(* Global variable list: TwinCAT_Configuration *)
(* Generated automatically by TwinCAT - (read only) *)
VAR_CONFIG
	ST_Hydra8.a_signal_produktion AT %QX228.0 : BOOL;
	ST_Hydra8.a_signal_gutteil AT %QX228.1 : BOOL;
	ST_Hydra8.a_signal_schlechtteil AT %QX228.2 : BOOL;
	ST_Hydra8.a_signal_reserve AT %QX228.3 : BOOL;
	.ST00_170_Motorschutz.BitInToCheck AT %IX1204.0 : BOOL;	(*  ~ {LinkedWith:TIID^Gerät 2 (EtherCAT)^251_A1 (EK1100)^251_A10 (EL1809)^Channel 15^.ST00_170_Motorschutz.BitInToCheck} *)
	.ST00_170_Thermokont.BitInToCheck AT %IX1204.1 : BOOL;	(*  ~ {LinkedWith:TIID^Gerät 2 (EtherCAT)^251_A1 (EK1100)^251_A10 (EL1809)^Channel 16^.ST00_170_Thermokont.BitInToCheck} *)
	.ST00_245_V1.BitOutToSet AT %QX256.0 : BOOL;
	.ST00_245_V1.BitInToCheck AT %IX1412.0 : BOOL;
	.ST00_245_V2_START.BitOutToSet AT %QX256.1 : BOOL;
	.ST00_245_V2_START.BitInToCheck AT %IX1412.1 : BOOL;
	.ST00_245_V3_RESET.BitOutToSet AT %QX256.2 : BOOL;
	.ST00_245_V3_RESET.BitInToCheck AT %IX1412.2 : BOOL;
	.ST00_245_S1_STOP.BitInToCheck AT %IX1412.3 : BOOL;
	.ST00_245_S2_START.BitInToCheck AT %IX1412.4 : BOOL;
	.ST00_245_S3_RESET.BitInToCheck AT %IX1412.5 : BOOL;
	.ST00_72_K7.BitOutToSet AT %QX128.0 : BOOL;	(*  ~ {LinkedWith:TIID^Gerät 2 (EtherCAT)^251_A1 (EK1100)^252_A21 (EL2809)^Channel 4^.ST00_72_K7.BitOutToSet} *)
	.ST00_72_K7.BitInToCheck AT %IX1240.0 : BOOL;
	.ST00_73_K4.BitInToCheck AT %IX1388.0 : BOOL;	(*  ~ {LinkedWith:TIID^Gerät 2 (EtherCAT)^S1 A1 (EK1101)^DI1 (EL1004)^Channel 3^.ST00_73_K4.BitInToCheck AND.ST02_S1_40K01.BitInToCheck} *)
	.ST02_DT_95_A1.e_Ergebnis_iO AT %IX1240.2 : BOOL;	(*  ~ {LinkedWith:TIID^Gerät 2 (EtherCAT)^S1 A1 (EK1101)^DI4  (EL1809)^Channel 11^.ST02_DT_95_A1.e_Ergebnis_iO} *)
	.ST02_DT_95_A1.e_Ergebnis_niO AT %IX1240.3 : BOOL;	(*  ~ {LinkedWith:TIID^Gerät 2 (EtherCAT)^S1 A1 (EK1101)^DI4  (EL1809)^Channel 10^.ST02_DT_95_A1.e_Ergebnis_niO} *)
	.ST02_DT_95_A1.e_Betriebsbereit AT %IX1240.4 : BOOL;	(*  ~ {LinkedWith:TIID^Gerät 2 (EtherCAT)^S1 A1 (EK1101)^DI4  (EL1809)^Channel 9^.ST02_DT_95_A1.e_Betriebsbereit} *)
	.ST02_DT_95_A1.e_Best_Jobwechsel AT %IX1240.5 : BOOL;
	.ST02_DT_95_A1.a_Trigger AT %QX128.2 : BOOL;	(*  ~ {LinkedWith:TIID^Gerät 2 (EtherCAT)^S1 A1 (EK1101)^DO3 (EL2809)^Channel 6^.ST02_DT_95_A1.a_Trigger} *)
	.ST02_DT_95_A1.a_Job_Bit1 AT %QX128.3 : BOOL;	(*  ~ {LinkedWith:TIID^Gerät 2 (EtherCAT)^S1 A1 (EK1101)^DO3 (EL2809)^Channel 7^.ST02_DT_95_A1.a_Job_Bit1} *)
	.ST02_DT_95_A1.a_Job_Bit2 AT %QX128.4 : BOOL;	(*  ~ {LinkedWith:TIID^Gerät 2 (EtherCAT)^S1 A1 (EK1101)^DO3 (EL2809)^Channel 8^.ST02_DT_95_A1.a_Job_Bit2} *)
	.ST02_DT_95_A1.a_Job_Bit3 AT %QX196.0 : BOOL;
	.ST02_DT_95_A1.a_Job_Bit4 AT %QX196.1 : BOOL;
	.ST02_DT_95_A2.e_Betriebsbereit AT %IX1340.0 : BOOL;	(*  ~ {LinkedWith:TIID^Gerät 2 (EtherCAT)^S1 A1 (EK1101)^DI4  (EL1809)^Channel 9^.ST02_DT_95_A1.e_Betriebsbereit} *)
	.ST02_S1_66_B11.ValveSensor AT %IX1260.0 : BOOL;	(*  ~ {LinkedWith:TIID^Gerät 2 (EtherCAT)^DT_61A1(EP1816-0008)^DIG Inputs Channel 2^.ST02_S1_66_B11.ValveSensor} *)
	.ST02_S1_66_B21.ValveSensor AT %IX1260.1 : BOOL;	(*  ~ {LinkedWith:TIID^Gerät 2 (EtherCAT)^DT_61A1(EP1816-0008)^DIG Inputs Channel 2^.ST02_S1_66_B21.ValveSensor} *)
	.ST02_S1_66_B31.ValveSensor AT %IX1260.2 : BOOL;	(*  ~ {LinkedWith:TIID^Gerät 2 (EtherCAT)^DT_61A1(EP1816-0008)^DIG Inputs Channel 2^.ST02_S1_66_B31.ValveSensor} *)
	.ST02_S1_66_B41.ValveSensor AT %IX1260.3 : BOOL;	(*  ~ {LinkedWith:TIID^Gerät 2 (EtherCAT)^DT_61A1(EP1816-0008)^DIG Inputs Channel 2^.ST02_S1_66_B41.ValveSensor} *)
	.ST02_FDB_40_B61.BitInToCheck AT %IX1308.0 : BOOL;	(*  ~ {LinkedWith:TIID^Gerät 2 (EtherCAT)^S1 A1 (EK1101)^DI2 (EL1004)^Channel 1^.ST02_FDB_40_B61.BitInToCheck} *)
	.ST02_FDB_40_B71.BitInToCheck AT %IX1308.1 : BOOL;	(*  ~ {LinkedWith:TIID^Gerät 2 (EtherCAT)^S1 A1 (EK1101)^DI2 (EL1004)^Channel 2^.ST02_FDB_40_B71.BitInToCheck} *)
	.ST02_35_S31.BitInToCheck AT %IX1244.0 : BOOL;	(*  ~ {LinkedWith:TIID^Gerät 2 (EtherCAT)^S1 A1 (EK1101)^DI3 (EL1004)^Channel 4^.ST02_35_S31.BitInToCheck} *)
	.ST02_S1_6A01.BitInToCheck AT %IX1256.0 : BOOL;	(*  ~ {LinkedWith:TIID^Gerät 2 (EtherCAT)^S1 A1 (EK1101)^DI1 (EL1004)^Channel 1^.ST02_S1_6A01.BitInToCheck} *)
	.ST02_35Y01.CoilA AT %QX136.0 : BOOL;	(*  ~ {LinkedWith:TIID^Gerät 2 (EtherCAT)^S1 A1 (EK1101)^DO2 (EL2004)^Channel 1^.ST02_35Y01.CoilA} *)
	.ST02_35Y01.CoilB AT %QX136.1 : BOOL;
	.ST02_62_Y6.CoilA AT %QX148.0 : BOOL;	(*  ~ {LinkedWith:TIID^Gerät 2 (EtherCAT)^TDA_61A1 (CPX-FB38 64Byte)^Outputs^QB0^.ST02_62_Y6.CoilA} *)
	.ST02_62_Y6.CoilB AT %QX148.1 : BOOL;	(*  ~ {LinkedWith:TIID^Gerät 2 (EtherCAT)^TDA_61A1 (CPX-FB38 64Byte)^Outputs^QB0^.ST02_62_Y6.CoilB} *)
	.ST02_62_Y9.CoilA AT %QX144.0 : BOOL;	(*  ~ {LinkedWith:TIID^Gerät 2 (EtherCAT)^TDA_61A1 (CPX-FB38 64Byte)^Outputs^QB1^.ST02_62_Y9.CoilA} *)
	.ST02_62_Y9.CoilB AT %QX144.1 : BOOL;	(*  ~ {LinkedWith:TIID^Gerät 2 (EtherCAT)^TDA_61A1 (CPX-FB38 64Byte)^Outputs^QB1^.ST02_62_Y9.CoilB} *)
	.ST02_62_Y11.CoilA AT %QX144.2 : BOOL;	(*  ~ {LinkedWith:TIID^Gerät 2 (EtherCAT)^TDA_61A1 (CPX-FB38 64Byte)^Outputs^QB1^.ST02_62_Y11.CoilA} *)
	.ST02_62_Y11.CoilB AT %QX144.3 : BOOL;	(*  ~ {LinkedWith:TIID^Gerät 2 (EtherCAT)^TDA_61A1 (CPX-FB38 64Byte)^Outputs^QB1^.ST02_62_Y11.CoilB} *)
	.ST02_62_Y13.CoilA AT %QX144.4 : BOOL;	(*  ~ {LinkedWith:TIID^Gerät 2 (EtherCAT)^TDA_61A1 (CPX-FB38 64Byte)^Outputs^QB1^.ST02_62_Y13.CoilA} *)
	.ST02_62_Y13.CoilB AT %QX144.5 : BOOL;	(*  ~ {LinkedWith:TIID^Gerät 2 (EtherCAT)^TDA_61A1 (CPX-FB38 64Byte)^Outputs^QB1^.ST02_62_Y13.CoilB} *)
	.ST02_62_Y15.CoilA AT %QX144.6 : BOOL;	(*  ~ {LinkedWith:TIID^Gerät 2 (EtherCAT)^TDA_61A1 (CPX-FB38 64Byte)^Outputs^QB1^.ST02_62_Y15.CoilA} *)
	.ST02_62_Y15.CoilB AT %QX144.7 : BOOL;	(*  ~ {LinkedWith:TIID^Gerät 2 (EtherCAT)^TDA_61A1 (CPX-FB38 64Byte)^Outputs^QB1^.ST02_62_Y15.CoilB} *)
	.ST02_62_Y17.CoilA AT %QX145.0 : BOOL;	(*  ~ {LinkedWith:TIID^Gerät 2 (EtherCAT)^TDA_61A1 (CPX-FB38 64Byte)^Outputs^QB2^.ST02_62_Y17.CoilA} *)
	.ST02_62_Y17.CoilB AT %QX145.1 : BOOL;
	.ST02_62_Y18.CoilA AT %QX145.2 : BOOL;	(*  ~ {LinkedWith:TIID^Gerät 2 (EtherCAT)^TDA_61A1 (CPX-FB38 64Byte)^Outputs^QB2^.ST02_62_Y18.CoilA} *)
	.ST02_62_Y18.CoilB AT %QX145.3 : BOOL;
	.ST03_51_M1.e_Position AT %IB1312 : UDINT;	(*  ~ {LinkedWith:TIID^Gerät 2 (EtherCAT)^251_A1 (EK1100)^252_PM1(EL7211-0010)^FB Position^.ST03_51_M1.e_Position} *)
	.ST03_51_M1.e_Statusword AT %IB1316 : UINT;	(*  ~ {LinkedWith:TIID^Gerät 2 (EtherCAT)^251_A1 (EK1100)^252_PM1(EL7211-0010)^DRV Statusword^.ST03_51_M1.e_Statusword} *)
	.ST03_51_M1.e_Velocity AT %IB1318 : DINT;	(*  ~ {LinkedWith:TIID^Gerät 2 (EtherCAT)^251_A1 (EK1100)^252_PM1(EL7211-0010)^DRV Velocity actual value^.ST03_51_M1.e_Velocity} *)
	.ST03_51_M1.e_Torque AT %IB1328 : INT;
	.ST03_51_M1.e_Following_Error AT %IB1322 : DINT;	(*  ~ {LinkedWith:TIID^Gerät 2 (EtherCAT)^251_A1 (EK1100)^252_PM1(EL7211-0010)^DRV Following error actual value^.ST03_51_M1.e_Following_Error} *)
	.ST03_51_M1.e_Toggle AT %IX1326.0 : BOOL;	(*  ~ {LinkedWith:TIID^Gerät 2 (EtherCAT)^251_A1 (EK1100)^252_PM1(EL7211-0010)^WcState^InputToggle} *)
	.ST03_51_M1.e_State AT %IB1377 : UINT;
	.ST03_51_M1.a_Controlword AT %QB176 : UINT;	(*  ~ {LinkedWith:TIID^Gerät 2 (EtherCAT)^251_A1 (EK1100)^252_PM1(EL7211-0010)^DRV Controlword^.ST03_51_M1.a_Controlword} *)
	.ST03_51_M1.a_Target_Velocity AT %QB178 : DINT;	(*  ~ {LinkedWith:TIID^Gerät 2 (EtherCAT)^251_A1 (EK1100)^252_PM1(EL7211-0010)^DRV Target velocity^.ST03_51_M1.a_Target_Velocity} *)
	.ST03_51_M1.a_Target_Position AT %QB182 : UDINT;	(*  ~ {LinkedWith:TIID^Gerät 2 (EtherCAT)^251_A1 (EK1100)^252_PM1(EL7211-0010)^DRV Target position^.ST03_51_M1.a_Target_Position} *)
	.ST03_601V1_A1.BitOutToSet AT %QX228.4 : BOOL;
	.ST03_601V1_A1.BitInToCheck AT %IX1379.0 : BOOL;
	.Robot01.CollisionSensor AT %IX1379.1 : BOOL;
	.ST03_BG3_X53_0.BitInToCheck AT %IX1340.1 : BOOL;
	.ST03_65_Q1.BitOutToSet AT %QX252.0 : BOOL;
	.ST03_65_Q1.BitInToCheck AT %IX1408.0 : BOOL;
	.ST03_65_F1.BitInToCheck AT %IX1408.1 : BOOL;
	.ST03_8_100_A1.e_Betriebsbereit AT %IX1412.6 : BOOL;
	.ST03_8_103_A1.e_Betriebsbereit AT %IX1480.0 : BOOL;
	.ST03_418_B60_0.ValveSensor AT %IX1296.0 : BOOL;
	.ST03_418_B60_1.ValveSensor AT %IX1296.1 : BOOL;
	.ST03_418_B60_2.ValveSensor AT %IX1296.2 : BOOL;
	.ST03_418_B60_3.ValveSensor AT %IX1296.3 : BOOL;
	.ST03_418_B60_4.ValveSensor AT %IX1296.4 : BOOL;
	.ST03_418_B60_5.ValveSensor AT %IX1296.5 : BOOL;
	.ST03_418_B60_6.BitInToCheck AT %IX1296.6 : BOOL;
	.ST03_418_B60_7.BitInToCheck AT %IX1296.7 : BOOL;
	.ST03_419_B61_0.BitInToCheck AT %IX1297.0 : BOOL;
	.ST03_419_B61_1.BitInToCheck AT %IX1297.1 : BOOL;
	.ST03_419_B61_2.BitInToCheck AT %IX1297.2 : BOOL;
	.ST03_419_B61_3.BitInToCheck AT %IX1297.3 : BOOL;
	.ST03_419_Y61_5.CoilA AT %QX172.0 : BOOL;
	.ST03_419_Y61_5.CoilB AT %QX172.1 : BOOL;
	.ST03_419_Y61_6.CoilA AT %QX172.2 : BOOL;
	.ST03_419_Y61_6.CoilB AT %QX172.3 : BOOL;
	.ST03_419_Y61_7.CoilA AT %QX172.4 : BOOL;
	.ST03_419_Y61_7.CoilB AT %QX172.5 : BOOL;
	.ST03_425_B67_0.ValveSensor AT %IX1330.0 : BOOL;
	.ST03_425_B67_1.ValveSensor AT %IX1330.1 : BOOL;
	.ST03_425_B67_2.ValveSensor AT %IX1330.2 : BOOL;
	.ST03_425_B67_3.ValveSensor AT %IX1330.3 : BOOL;
	.ST03_425_B67_4.BitInToCheck AT %IX1330.4 : BOOL;
	.ST03_425_B67_5.BitInToCheck AT %IX1330.5 : BOOL;
	.ST03_425_B67_6.BitInToCheck AT %IX1330.6 : BOOL;
	.ST03_425_B67_7.BitInToCheck AT %IX1330.7 : BOOL;
	.ST03_426_B68_4.BitInToCheck AT %IX1331.0 : BOOL;
	.ST03_426_Y68_5.CoilA AT %QX188.0 : BOOL;
	.ST03_426_Y68_5.CoilB AT %QX188.1 : BOOL;
	.ST03_426_Y68_6.CoilA AT %QX188.2 : BOOL;
	.ST03_426_Y68_6.CoilB AT %QX188.3 : BOOL;
	.ST03_421_B63_0.ValveSensor AT %IX1297.4 : BOOL;
	.ST03_421_B63_1.ValveSensor AT %IX1297.5 : BOOL;
	.ST03_421_B63_2.ValveSensor AT %IX1297.6 : BOOL;
	.ST03_421_B63_3.ValveSensor AT %IX1297.7 : BOOL;
	.ST03_421_B63_4.BitInToCheck AT %IX1298.0 : BOOL;
	.ST03_421_B63_5.BitInToCheck AT %IX1298.1 : BOOL;
	.ST03_421_B63_6.BitInToCheck AT %IX1298.2 : BOOL;
	.ST03_421_B63_7.BitInToCheck AT %IX1298.3 : BOOL;
	.ST03_422_B64_0.BitInToCheck AT %IX1298.4 : BOOL;
	.ST03_423_B66_0.BitInToCheck AT %IX1340.2 : BOOL;
	.ST03_8_B76_1.BitInToCheck AT %IX1340.3 : BOOL;
	.ST03_8_B76_2.BitInToCheck AT %IX1340.4 : BOOL;
	.ST03_422_B64_1.ValveSensor AT %IX1298.5 : BOOL;
	.ST03_422_B64_2.ValveSensor AT %IX1298.6 : BOOL;
	.ST03_422_B64_3.BitInToCheck AT %IX1298.7 : BOOL;
	.ST03_422_B64_4.BitInToCheck AT %IX1299.0 : BOOL;
	.ST03_422_Y64_5.CoilA AT %QX172.6 : BOOL;
	.ST03_422_Y64_5.CoilB AT %QX172.7 : BOOL;
	.ST03_422_Y64_6.CoilA AT %QX173.0 : BOOL;
	.ST03_422_Y64_6.CoilB AT %QX173.1 : BOOL;
	.ST03_422_Y64_7.CoilA AT %QX173.2 : BOOL;
	.ST03_422_Y64_7.CoilB AT %QX173.3 : BOOL;
	.ST03_423_B65_0.ValveSensor AT %IX1340.5 : BOOL;
	.ST03_423_B65_1.ValveSensor AT %IX1340.6 : BOOL;
	.ST03_423_B65_2.BitInToCheck AT %IX1340.7 : BOOL;
	.ST03_423_B65_3.ValveSensor AT %IX1341.0 : BOOL;
	.ST03_423_B65_4.ValveSensor AT %IX1341.1 : BOOL;
	.ST03_423_B65_5.BitInToCheck AT %IX1341.2 : BOOL;
	.ST03_423_Y65_6.CoilA AT %QX196.2 : BOOL;
	.ST03_423_Y65_6.CoilB AT %QX196.3 : BOOL;
	.ST03_423_Y65_7.CoilA AT %QX196.4 : BOOL;
	.ST03_423_Y65_7.CoilB AT %QX196.5 : BOOL;
	.ST03_33F4.BitInToCheck AT %IX1299.1 : BOOL;
	.ST03_70U3_1.BitInToCheck AT %IX1299.2 : BOOL;
	.ST03_70U3_2.BitInToCheck AT %IX1299.3 : BOOL;
	.ST03_70U3_3.BitInToCheck AT %IX1299.4 : BOOL;
	.ST03_71U3_1.BitInToCheck AT %IX1299.5 : BOOL;
	.ST03_71U3_2.BitInToCheck AT %IX1299.6 : BOOL;
	.ST03_71U3_3.BitInToCheck AT %IX1299.7 : BOOL;
	.ST03_8_80_A1.e_Ergebnis_iO AT %IX1300.0 : BOOL;
	.ST03_8_80_A1.e_Ergebnis_niO AT %IX1300.1 : BOOL;
	.ST03_8_80_A1.e_Betriebsbereit AT %IX1300.2 : BOOL;
	.ST03_8_80_A1.e_Best_Jobwechsel AT %IX1300.3 : BOOL;
	.ST03_8_80_A1.a_Trigger AT %QX173.4 : BOOL;
	.ST03_8_80_A1.a_Job_Bit1 AT %QX173.5 : BOOL;
	.ST03_8_80_A1.a_Job_Bit2 AT %QX173.6 : BOOL;
	.ST03_8_80_A1.a_Job_Bit3 AT %QX196.6 : BOOL;
	.ST03_8_80_A1.a_Job_Bit4 AT %QX196.7 : BOOL;
	.ST03_8_85_A1.e_Ergebnis_iO AT %IX1300.4 : BOOL;
	.ST03_8_85_A1.e_Ergebnis_niO AT %IX1300.5 : BOOL;
	.ST03_8_85_A1.e_Betriebsbereit AT %IX1300.6 : BOOL;
	.ST03_8_85_A1.e_Best_Jobwechsel AT %IX1300.7 : BOOL;
	.ST03_8_85_A1.a_Trigger AT %QX173.7 : BOOL;
	.ST03_8_85_A1.a_Job_Bit1 AT %QX174.0 : BOOL;
	.ST03_8_85_A1.a_Job_Bit2 AT %QX174.1 : BOOL;
	.ST03_8_85_A1.a_Job_Bit3 AT %QX197.0 : BOOL;
	.ST03_8_85_A1.a_Job_Bit4 AT %QX197.1 : BOOL;
	.ST03_8_90_A1.e_Betriebsbereit AT %IX1341.3 : BOOL;
	.ST03_8_95_A1.e_Betriebsbereit AT %IX1341.4 : BOOL;
	.ST03_PLAN_70V1_1.BitOutToSet AT %QX174.2 : BOOL;
	.ST03_PLAN_70V1_1.BitInToCheck AT %IX1301.0 : BOOL;
	.ST03_PLAN_71V1_2.BitOutToSet AT %QX174.3 : BOOL;
	.ST03_PLAN_71V1_2.BitInToCheck AT %IX1301.1 : BOOL;
	.ST03_Y01.CoilA AT %QX197.2 : BOOL;
	.ST03_Y01.CoilB AT %QX197.3 : BOOL;
	.ST03_S18.BitInToCheck AT %IX1341.5 : BOOL;
	.ST03_435_B67_0.ValveSensor AT %IX1336.0 : BOOL;
	.ST03_435_B67_1.ValveSensor AT %IX1336.1 : BOOL;
	.ST03_435_B67_2.ValveSensor AT %IX1336.2 : BOOL;
	.ST03_435_B67_3.ValveSensor AT %IX1336.3 : BOOL;
	.ST03_435_B67_4.BitInToCheck AT %IX1336.4 : BOOL;
	.ST03_435_B67_7.BitInToCheck AT %IX1336.5 : BOOL;
	.ST03_436_B68_1.BitInToCheck AT %IX1336.6 : BOOL;
	.ST03_436_B68_2.BitInToCheck AT %IX1336.7 : BOOL;
	.ST03_437_B68_3.BitInToCheck AT %IX1337.0 : BOOL;
	.ST03_437_B68_4.BitInToCheck AT %IX1337.1 : BOOL;
	.ST03_437_Y68_5.CoilA AT %QX192.0 : BOOL;
	.ST03_437_Y68_5.CoilB AT %QX192.1 : BOOL;
	.ST03_437_Y68_6.CoilA AT %QX192.2 : BOOL;
	.ST03_437_Y68_6.CoilB AT %QX192.3 : BOOL;
	.ST03_444_B69_0.ValveSensor AT %IX1341.6 : BOOL;
	.ST03_444_B69_1.ValveSensor AT %IX1341.7 : BOOL;
	.ST03_444_B69_2.ValveSensor AT %IX1342.0 : BOOL;
	.ST03_444_B69_3.ValveSensor AT %IX1342.1 : BOOL;
	.ST03_444_B69_4.BitInToCheck AT %IX1342.2 : BOOL;
	.ST03_444_B69_7.BitInToCheck AT %IX1342.3 : BOOL;
	.ST03_445_B70_1.BitInToCheck AT %IX1342.4 : BOOL;
	.ST03_445_B70_2.BitInToCheck AT %IX1342.5 : BOOL;
	.ST03_446_B70_3.BitInToCheck AT %IX1342.6 : BOOL;
	.ST03_446_B70_4.BitInToCheck AT %IX1342.7 : BOOL;
	.ST03_446_Y70_5.CoilA AT %QX197.4 : BOOL;
	.ST03_446_Y70_5.CoilB AT %QX197.5 : BOOL;
	.ST03_446_Y70_6.CoilA AT %QX197.6 : BOOL;
	.ST03_446_Y70_6.CoilB AT %QX197.7 : BOOL;
	.ST03_451_B69_0.ValveSensor AT %IX1344.0 : BOOL;
	.ST03_451_B69_1.ValveSensor AT %IX1344.1 : BOOL;
	.ST03_451_B69_2.ValveSensor AT %IX1344.2 : BOOL;
	.ST03_451_B69_3.ValveSensor AT %IX1344.3 : BOOL;
	.ST03_451_B69_4.BitInToCheck AT %IX1344.4 : BOOL;
	.ST03_451_B69_7.BitInToCheck AT %IX1344.5 : BOOL;
	.ST03_452_B70_1.BitInToCheck AT %IX1344.6 : BOOL;
	.ST03_452_B70_2.BitInToCheck AT %IX1344.7 : BOOL;
	.ST03_453_B70_3.BitInToCheck AT %IX1345.0 : BOOL;
	.ST03_453_B70_4.BitInToCheck AT %IX1345.1 : BOOL;
	.ST03_453_Y70_5.CoilA AT %QX204.0 : BOOL;
	.ST03_453_Y70_5.CoilB AT %QX204.1 : BOOL;
	.ST03_453_Y70_6.CoilA AT %QX204.2 : BOOL;
	.ST03_453_Y70_6.CoilB AT %QX204.3 : BOOL;
	.ST03_461_B69_0.ValveSensor AT %IX1364.1 : BOOL;
	.ST03_461_B69_1.ValveSensor AT %IX1364.2 : BOOL;
	.ST03_461_B69_2.ValveSensor AT %IX1364.3 : BOOL;
	.ST03_461_B69_3.ValveSensor AT %IX1364.4 : BOOL;
	.ST03_461_B69_4.BitInToCheck AT %IX1364.5 : BOOL;
	.ST03_461_B69_5.ValveSensor AT %IX1364.6 : BOOL;
	.ST03_461_B69_6.ValveSensor AT %IX1364.7 : BOOL;
	.ST03_461_B69_7.BitInToCheck AT %IX1365.0 : BOOL;
	.ST03_462_B70_0.BitInToCheck AT %IX1365.1 : BOOL;
	.ST03_462_B70_1.BitInToCheck AT %IX1365.2 : BOOL;
	.ST03_462_B70_2.BitInToCheck AT %IX1365.3 : BOOL;
	.ST03_463_B70_3.ValveSensor AT %IX1365.4 : BOOL;
	.ST03_463_B70_4.ValveSensor AT %IX1365.5 : BOOL;
	.ST03_463_B70_5.ValveSensor AT %IX1365.6 : BOOL;
	.ST03_463_B70_6.ValveSensor AT %IX1365.7 : BOOL;
	.ST03_463_B70_7.BitInToCheck AT %IX1366.0 : BOOL;
	.ST03_464_Y71_0.CoilA AT %QX218.0 : BOOL;
	.ST03_464_Y71_0.CoilB AT %QX218.1 : BOOL;
	.ST03_464_Y71_1.CoilA AT %QX218.2 : BOOL;
	.ST03_464_Y71_1.CoilB AT %QX218.3 : BOOL;
	.ST03_464_Y71_2.CoilA AT %QX218.4 : BOOL;
	.ST03_464_Y71_2.CoilB AT %QX218.5 : BOOL;
	.ST03_464_Y71_3.CoilA AT %QX218.6 : BOOL;
	.ST03_464_Y71_3.CoilB AT %QX218.7 : BOOL;
	.ST03_464_Y71_4.CoilA AT %QX219.0 : BOOL;
	.ST03_464_Y71_4.CoilB AT %QX219.1 : BOOL;
	.ST03_464_Y71_5.CoilA AT %QX219.2 : BOOL;
	.ST03_464_Y71_5.CoilB AT %QX219.3 : BOOL;
	.ST03_464_B71_6.BitInToCheck AT %IX1366.1 : BOOL;
	.ST03_464_B71_7.BitInToCheck AT %IX1366.2 : BOOL;
	.ST03_8_105_A1.anInputRequest AT %QB288 : ARRAY [0..4] OF DWORD;
	.ST03_8_105_A1.bError_Status_00 AT %IX1464.0 : BOOL;
	.ST03_8_105_A1.bChange_Program_Ack AT %IX1464.1 : BOOL;
	.ST03_8_105_A1.bChange_Program_Failed AT %IX1464.2 : BOOL;
	.ST03_8_105_A1.bTotal_Status_OK_01 AT %IX1464.3 : BOOL;
	.ST03_8_105_A1.bTotal_Status_NG AT %IX1464.4 : BOOL;
	.ST03_8_105_A1.bRun AT %IX1464.5 : BOOL;
	.ST03_8_105_A1.bBusy AT %IX1464.6 : BOOL;
	.ST03_8_105_A1.bTrigger_Ready AT %IX1464.7 : BOOL;
	.ST03_8_105_A1.bTrigger_Ack AT %IX1465.0 : BOOL;
	.ST03_8_105_A1.abProgram_Num AT %IB1466 : ARRAY [0..6] OF BOOL;
	.ST03_8_105_A1.nState AT %IB1473 : UINT;
	.ST03_4x2_B69_0.BitInToCheck AT %IX1366.3 : BOOL;
	.ST03_4x2_B69_1.ValveSensor AT %IX1366.4 : BOOL;
	.ST03_4x2_B69_2.ValveSensor AT %IX1366.5 : BOOL;
	.ST03_4x2_B69_3.ValveSensor AT %IX1366.6 : BOOL;
	.ST03_4x2_B69_4.ValveSensor AT %IX1366.7 : BOOL;
	.ST03_4x2_B69_5.BitInToCheck AT %IX1392.0 : BOOL;
	.ST03_4x2_B69_6.ValveSensor AT %IX1367.1 : BOOL;
	.ST03_4x2_B69_7.ValveSensor AT %IX1392.1 : BOOL;
	.ST03_4x3_B70_0.BitInToCheck AT %IX1367.3 : BOOL;
	.ST03_4x3_B70_1.BitInToCheck AT %IX1392.2 : BOOL;
	.ST03_4x3_Y70_5.CoilA AT %QX236.0 : BOOL;
	.ST03_4x3_Y70_5.CoilB AT %QX236.1 : BOOL;
	.ST03_4x3_Y70_6.CoilA AT %QX236.2 : BOOL;
	.ST03_4x3_Y70_6.CoilB AT %QX236.3 : BOOL;
	.ST03_4x3_Y70_7.CoilA AT %QX236.4 : BOOL;
	.ST03_4x3_Y70_7.CoilB AT %QX236.5 : BOOL;
	.ST03_491_B69_0.BitInToCheck AT %IX1372.0 : BOOL;
	.ST03_491_B69_1.ValveSensor AT %IX1372.1 : BOOL;
	.ST03_491_B69_2.ValveSensor AT %IX1372.2 : BOOL;
	.ST03_491_B69_3.ValveSensor AT %IX1372.3 : BOOL;
	.ST03_491_B69_4.ValveSensor AT %IX1372.4 : BOOL;
	.ST03_491_B69_5.BitInToCheck AT %IX1372.5 : BOOL;
	.ST03_491_B69_7.BitInToCheck AT %IX1372.6 : BOOL;
	.ST03_492_Y70_0.CoilA AT %QX224.0 : BOOL;
	.ST03_492_Y70_0.CoilB AT %QX224.1 : BOOL;
	.ST03_492_Y70_1.CoilA AT %QX224.2 : BOOL;
	.ST03_492_Y70_1.CoilB AT %QX224.3 : BOOL;
	.ST03_501_B69_0.BitInToCheck AT %IX1379.4 : BOOL;
	.ST03_501_B69_1.ValveSensor AT %IX1379.5 : BOOL;
	.ST03_501_B69_2.ValveSensor AT %IX1379.6 : BOOL;
	.ST03_501_B69_3.ValveSensor AT %IX1379.7 : BOOL;
	.ST03_501_B69_4.ValveSensor AT %IX1380.0 : BOOL;
	.ST03_501_B69_5.BitInToCheck AT %IX1380.1 : BOOL;
	.ST03_501_B69_6.BitInToCheck AT %IX1380.2 : BOOL;
	.ST03_501_B69_7.BitInToCheck AT %IX1380.3 : BOOL;
	.ST03_502_B70_0.BitInToCheck AT %IX1380.4 : BOOL;
	.ST03_502_Y70_1.CoilA AT %QX228.7 : BOOL;
	.ST03_502_Y70_1.CoilB AT %QX229.0 : BOOL;
	.ST03_502_Y70_2.CoilA AT %QX229.1 : BOOL;
	.ST03_502_Y70_2.CoilB AT %QX229.2 : BOOL;
	.ST03_521_B69_0.BitInToCheck AT %IX1392.3 : BOOL;
	.ST03_521_B69_1.ValveSensor AT %IX1392.4 : BOOL;
	.ST03_521_B69_2.ValveSensor AT %IX1392.5 : BOOL;
	.ST03_521_B69_3.ValveSensor AT %IX1392.6 : BOOL;
	.ST03_521_B69_4.ValveSensor AT %IX1392.7 : BOOL;
	.ST03_521_B69_6.BitInToCheck AT %IX1393.0 : BOOL;
	.ST03_521_B69_7.BitInToCheck AT %IX1393.1 : BOOL;
	.ST03_522_B70_0.BitInToCheck AT %IX1393.2 : BOOL;
	.ST03_522_Y70_1.CoilA AT %QX236.6 : BOOL;
	.ST03_522_Y70_1.CoilB AT %QX236.7 : BOOL;
	.ST03_522_Y70_2.CoilA AT %QX237.0 : BOOL;
	.ST03_522_Y70_2.CoilB AT %QX237.1 : BOOL;
	.ST03_512_XG1.BitInToCheck AT %IX1380.5 : BOOL;	(*  ~ {LinkedWith:TIID^Gerät 2 (EtherCAT)^930_A2 (EP2338-0001)^Channel 1^.ST03_512_XG1.BitInToCheck} *)
	.ST03_512_B69_1.ValveSensor AT %IX1380.6 : BOOL;	(*  ~ {LinkedWith:TIID^Gerät 2 (EtherCAT)^930_A2 (EP2338-0001)^Channel 2^.ST03_512_B69_1.ValveSensor} *)
	.ST03_512_B69_2.ValveSensor AT %IX1380.7 : BOOL;	(*  ~ {LinkedWith:TIID^Gerät 2 (EtherCAT)^930_A2 (EP2338-0001)^Channel 3^.ST03_512_B69_2.ValveSensor} *)
	.ST03_512_B69_3.ValveSensor AT %IX1381.0 : BOOL;	(*  ~ {LinkedWith:TIID^Gerät 2 (EtherCAT)^930_A2 (EP2338-0001)^Channel 4^.ST03_512_B69_3.ValveSensor} *)
	.ST03_512_B69_4.ValveSensor AT %IX1381.1 : BOOL;	(*  ~ {LinkedWith:TIID^Gerät 2 (EtherCAT)^930_A2 (EP2338-0001)^Channel 5^.ST03_512_B69_4.ValveSensor} *)
	.ST03_512_B69_5.ValveSensor AT %IX1388.1 : BOOL;	(*  ~ {LinkedWith:TIID^Gerät 2 (EtherCAT)^930_A2 (EP2338-0001)^Channel 6^.ST03_512_B69_5.ValveSensor} *)
	.ST03_512_B69_6.ValveSensor AT %IX1388.2 : BOOL;	(*  ~ {LinkedWith:TIID^Gerät 2 (EtherCAT)^930_A2 (EP2338-0001)^Channel 7^.ST03_512_B69_6.ValveSensor} *)
	.ST03_513_B70_0.ValveSensor AT %IX1381.3 : BOOL;	(*  ~ {LinkedWith:TIID^Gerät 2 (EtherCAT)^931_A3 (EP2338-0001)^Channel 1^.ST03_513_B70_0.ValveSensor} *)
	.ST03_513_B70_1.ValveSensor AT %IX1381.4 : BOOL;	(*  ~ {LinkedWith:TIID^Gerät 2 (EtherCAT)^931_A3 (EP2338-0001)^Channel 2^.ST03_513_B70_1.ValveSensor} *)
	.ST03_513_B70_2.ValveSensor AT %IX1381.5 : BOOL;	(*  ~ {LinkedWith:TIID^Gerät 2 (EtherCAT)^931_A3 (EP2338-0001)^Channel 3^.ST03_513_B70_2.ValveSensor} *)
	.ST03_513_B70_3.ValveSensor AT %IX1381.6 : BOOL;	(*  ~ {LinkedWith:TIID^Gerät 2 (EtherCAT)^931_A3 (EP2338-0001)^Channel 4^.ST03_513_B70_3.ValveSensor} *)
	.ST03_513_B70_4.BitInToCheck AT %IX1381.7 : BOOL;	(*  ~ {LinkedWith:TIID^Gerät 2 (EtherCAT)^931_A3 (EP2338-0001)^Channel 5^.ST03_513_B70_4.BitInToCheck} *)
	.ST03_513_B70_5.ValveSensor AT %IX1382.0 : BOOL;	(*  ~ {LinkedWith:TIID^Gerät 2 (EtherCAT)^931_A3 (EP2338-0001)^Channel 6^.ST03_513_B70_5.ValveSensor} *)
	.ST03_513_B70_6.ValveSensor AT %IX1382.1 : BOOL;	(*  ~ {LinkedWith:TIID^Gerät 2 (EtherCAT)^931_A3 (EP2338-0001)^Channel 7^.ST03_513_B70_6.ValveSensor} *)
	.ST03_513_B70_7.BitInToCheck AT %IX1382.2 : BOOL;	(*  ~ {LinkedWith:TIID^Gerät 2 (EtherCAT)^931_A3 (EP2338-0001)^Channel 8^.ST03_513_B70_7.BitInToCheck} *)
	.ST03_514_B71_0.ValveSensor AT %IX1382.3 : BOOL;	(*  ~ {LinkedWith:TIID^Gerät 2 (EtherCAT)^931_A4 (EP2338-0001)^Channel 1^.ST03_514_B71_0.ValveSensor} *)
	.ST03_514_B71_1.ValveSensor AT %IX1382.4 : BOOL;	(*  ~ {LinkedWith:TIID^Gerät 2 (EtherCAT)^931_A4 (EP2338-0001)^Channel 2^.ST03_514_B71_1.ValveSensor} *)
	.ST03_514_B71_2.BitInToCheck AT %IX1382.5 : BOOL;	(*  ~ {LinkedWith:TIID^Gerät 2 (EtherCAT)^931_A4 (EP2338-0001)^Channel 3^.ST03_514_B71_2.BitInToCheck} *)
	.ST03_514_B71_3.ValveSensor AT %IX1382.6 : BOOL;	(*  ~ {LinkedWith:TIID^Gerät 2 (EtherCAT)^931_A4 (EP2338-0001)^Channel 4^.ST03_514_B71_3.ValveSensor} *)
	.ST03_514_B71_4.ValveSensor AT %IX1382.7 : BOOL;	(*  ~ {LinkedWith:TIID^Gerät 2 (EtherCAT)^931_A4 (EP2338-0001)^Channel 5^.ST03_514_B71_4.ValveSensor} *)
	.ST03_514_B71_5.BitInToCheck AT %IX1383.0 : BOOL;	(*  ~ {LinkedWith:TIID^Gerät 2 (EtherCAT)^931_A4 (EP2338-0001)^Channel 6^.ST03_514_B71_5.BitInToCheck} *)
	.ST03_514_B71_6.BitInToCheck AT %IX1383.1 : BOOL;	(*  ~ {LinkedWith:TIID^Gerät 2 (EtherCAT)^931_A4 (EP2338-0001)^Channel 7^.ST03_514_B71_6.BitInToCheck} *)
	.ST03_514_B71_7.BitInToCheck AT %IX1388.3 : BOOL;	(*  ~ {LinkedWith:TIID^Gerät 2 (EtherCAT)^931_A4 (EP2338-0001)^Channel 8^.ST03_514_B71_7.BitInToCheck} *)
	.ST03_515_Y72_0.CoilA AT %QX232.0 : BOOL;	(*  ~ {LinkedWith:TIID^Gerät 2 (EtherCAT)^932_A5 (EP2338-0001)^Channel 9^.ST03_515_Y72_0.CoilA} *)
	.ST03_515_Y72_0.CoilB AT %QX232.1 : BOOL;
	.ST03_515_Y72_1.CoilA AT %QX232.2 : BOOL;	(*  ~ {LinkedWith:TIID^Gerät 2 (EtherCAT)^932_A5 (EP2338-0001)^Channel 10^.ST03_515_Y72_1.CoilA} *)
	.ST03_515_Y72_1.CoilB AT %QX232.3 : BOOL;
	.ST03_515_Y72_2.CoilA AT %QX232.4 : BOOL;	(*  ~ {LinkedWith:TIID^Gerät 2 (EtherCAT)^932_A5 (EP2338-0001)^Channel 11^.ST03_515_Y72_2.CoilA} *)
	.ST03_515_Y72_2.CoilB AT %QX232.5 : BOOL;
	.ST03_515_Y72_3.CoilA AT %QX232.6 : BOOL;	(*  ~ {LinkedWith:TIID^Gerät 2 (EtherCAT)^932_A5 (EP2338-0001)^Channel 12^.ST03_515_Y72_3.CoilA} *)
	.ST03_515_Y72_3.CoilB AT %QX232.7 : BOOL;
	.ST03_515_Y72_4.CoilA AT %QX233.0 : BOOL;	(*  ~ {LinkedWith:TIID^Gerät 2 (EtherCAT)^932_A5 (EP2338-0001)^Channel 13^.ST03_515_Y72_4.CoilA} *)
	.ST03_515_Y72_4.CoilB AT %QX233.1 : BOOL;
	.ST03_515_Y72_5.CoilA AT %QX233.2 : BOOL;	(*  ~ {LinkedWith:TIID^Gerät 2 (EtherCAT)^932_A5 (EP2338-0001)^Channel 14^.ST03_515_Y72_5.CoilA} *)
	.ST03_515_Y72_5.CoilB AT %QX233.3 : BOOL;
	.ST03_515_Y72_6.CoilA AT %QX233.4 : BOOL;	(*  ~ {LinkedWith:TIID^Gerät 2 (EtherCAT)^932_A5 (EP2338-0001)^Channel 15^.ST03_515_Y72_6.CoilA} *)
	.ST03_515_Y72_6.CoilB AT %QX233.5 : BOOL;
	.ST03_531_B69_0.BitInToCheck AT %IX1396.0 : BOOL;
	.ST03_531_B69_1.ValveSensor AT %IX1396.1 : BOOL;
	.ST03_531_B69_2.ValveSensor AT %IX1396.2 : BOOL;
	.ST03_531_B69_3.ValveSensor AT %IX1396.3 : BOOL;
	.ST03_531_B69_4.ValveSensor AT %IX1396.4 : BOOL;
	.ST03_531_B69_6.BitInToCheck AT %IX1396.5 : BOOL;
	.ST03_531_B69_7.BitInToCheck AT %IX1396.6 : BOOL;
	.ST03_532_B70_0.BitInToCheck AT %IX1396.7 : BOOL;
	.ST03_532_Y70_1.CoilA AT %QX240.0 : BOOL;
	.ST03_532_Y70_1.CoilB AT %QX240.1 : BOOL;
	.ST03_532_Y70_2.CoilA AT %QX240.2 : BOOL;
	.ST03_532_Y70_2.CoilB AT %QX240.3 : BOOL;
	.ST03_536_B69_0.BitInToCheck AT %IX1400.0 : BOOL;
	.ST03_536_B69_1.ValveSensor AT %IX1400.1 : BOOL;
	.ST03_536_B69_2.ValveSensor AT %IX1400.2 : BOOL;
	.ST03_536_B69_3.ValveSensor AT %IX1400.3 : BOOL;
	.ST03_536_B69_4.ValveSensor AT %IX1400.4 : BOOL;
	.ST03_536_B69_6.BitInToCheck AT %IX1400.5 : BOOL;
	.ST03_536_B69_7.BitInToCheck AT %IX1400.6 : BOOL;
	.ST03_537_B70_0.BitInToCheck AT %IX1400.7 : BOOL;
	.ST03_537_Y70_1.CoilA AT %QX244.0 : BOOL;
	.ST03_537_Y70_1.CoilB AT %QX244.1 : BOOL;
	.ST03_537_Y70_2.CoilA AT %QX244.2 : BOOL;
	.ST03_537_Y70_2.CoilB AT %QX244.3 : BOOL;
	.ST03_541_B69_0.BitInToCheck AT %IX1404.0 : BOOL;
	.ST03_541_B69_1.ValveSensor AT %IX1404.1 : BOOL;
	.ST03_541_B69_2.ValveSensor AT %IX1404.2 : BOOL;
	.ST03_541_B69_3.ValveSensor AT %IX1404.3 : BOOL;
	.ST03_541_B69_4.ValveSensor AT %IX1404.4 : BOOL;
	.ST03_541_B69_6.BitInToCheck AT %IX1404.5 : BOOL;
	.ST03_541_B69_7.BitInToCheck AT %IX1404.6 : BOOL;
	.ST03_542_B70_0.BitInToCheck AT %IX1404.7 : BOOL;
	.ST03_542_Y70_1.CoilA AT %QX248.0 : BOOL;
	.ST03_542_Y70_1.CoilB AT %QX248.1 : BOOL;
	.ST03_542_Y70_2.CoilA AT %QX248.2 : BOOL;
	.ST03_542_Y70_2.CoilB AT %QX248.3 : BOOL;
	.ST03_546_B69_0.BitInToCheck AT %IX1405.0 : BOOL;	(*  ~ {LinkedWith:TIID^Gerät 2 (EtherCAT)^945_A2 (EP2338-0001)^Channel 1^.ST03_546_B69_0.BitInToCheck} *)
	.ST03_546_B69_1.ValveSensor AT %IX1405.1 : BOOL;	(*  ~ {LinkedWith:TIID^Gerät 2 (EtherCAT)^945_A2 (EP2338-0001)^Channel 2^.ST03_546_B69_1.ValveSensor} *)
	.ST03_546_B69_2.ValveSensor AT %IX1405.2 : BOOL;	(*  ~ {LinkedWith:TIID^Gerät 2 (EtherCAT)^945_A2 (EP2338-0001)^Channel 3^.ST03_546_B69_2.ValveSensor} *)
	.ST03_546_B69_3.ValveSensor AT %IX1405.3 : BOOL;	(*  ~ {LinkedWith:TIID^Gerät 2 (EtherCAT)^945_A2 (EP2338-0001)^Channel 4^.ST03_546_B69_3.ValveSensor} *)
	.ST03_546_B69_4.ValveSensor AT %IX1405.4 : BOOL;	(*  ~ {LinkedWith:TIID^Gerät 2 (EtherCAT)^945_A2 (EP2338-0001)^Channel 5^.ST03_546_B69_4.ValveSensor} *)
	.ST03_546_B69_6.BitInToCheck AT %IX1405.5 : BOOL;	(*  ~ {LinkedWith:TIID^Gerät 2 (EtherCAT)^945_A2 (EP2338-0001)^Channel 7^.ST03_546_B69_6.BitInToCheck} *)
	.ST03_546_B69_7.BitInToCheck AT %IX1405.6 : BOOL;	(*  ~ {LinkedWith:TIID^Gerät 2 (EtherCAT)^945_A2 (EP2338-0001)^Channel 8^.ST03_546_B69_7.BitInToCheck} *)
	.ST03_547_B70_0.BitInToCheck AT %IX1405.7 : BOOL;	(*  ~ {LinkedWith:TIID^Gerät 2 (EtherCAT)^945_A3 (EP2338-0001)^Channel 1^.ST03_547_B70_0.BitInToCheck} *)
	.ST03_547_Y70_1.CoilA AT %QX248.4 : BOOL;	(*  ~ {LinkedWith:TIID^Gerät 2 (EtherCAT)^945_A3 (EP2338-0001)^Channel 10^.ST03_547_Y70_1.CoilA} *)
	.ST03_547_Y70_1.CoilB AT %QX248.5 : BOOL;
	.ST03_547_Y70_2.CoilA AT %QX248.6 : BOOL;	(*  ~ {LinkedWith:TIID^Gerät 2 (EtherCAT)^945_A3 (EP2338-0001)^Channel 11^.ST03_547_Y70_2.CoilA} *)
	.ST03_547_Y70_2.CoilB AT %QX248.7 : BOOL;
	.ST03_551_B69_0.BitInToCheck AT %IX1406.0 : BOOL;	(*  ~ {LinkedWith:TIID^Gerät 2 (EtherCAT)^946_A2 (EP2338-0001)^Channel 1^.ST03_551_B69_0.BitInToCheck} *)
	.ST03_551_B69_1.ValveSensor AT %IX1406.1 : BOOL;	(*  ~ {LinkedWith:TIID^Gerät 2 (EtherCAT)^946_A2 (EP2338-0001)^Channel 2^.ST03_551_B69_1.ValveSensor} *)
	.ST03_551_B69_2.ValveSensor AT %IX1406.2 : BOOL;	(*  ~ {LinkedWith:TIID^Gerät 2 (EtherCAT)^946_A2 (EP2338-0001)^Channel 3^.ST03_551_B69_2.ValveSensor} *)
	.ST03_551_B69_3.ValveSensor AT %IX1406.3 : BOOL;	(*  ~ {LinkedWith:TIID^Gerät 2 (EtherCAT)^946_A2 (EP2338-0001)^Channel 4^.ST03_551_B69_3.ValveSensor} *)
	.ST03_551_B69_4.ValveSensor AT %IX1406.4 : BOOL;	(*  ~ {LinkedWith:TIID^Gerät 2 (EtherCAT)^946_A2 (EP2338-0001)^Channel 5^.ST03_551_B69_4.ValveSensor} *)
	.ST03_551_B69_6.BitInToCheck AT %IX1406.5 : BOOL;	(*  ~ {LinkedWith:TIID^Gerät 2 (EtherCAT)^946_A2 (EP2338-0001)^Channel 7^.ST03_551_B69_6.BitInToCheck} *)
	.ST03_551_B69_7.BitInToCheck AT %IX1406.6 : BOOL;	(*  ~ {LinkedWith:TIID^Gerät 2 (EtherCAT)^946_A2 (EP2338-0001)^Channel 8^.ST03_551_B69_7.BitInToCheck} *)
	.ST03_552_B70_0.BitInToCheck AT %IX1406.7 : BOOL;	(*  ~ {LinkedWith:TIID^Gerät 2 (EtherCAT)^946_A3 (EP2338-0001)^Channel 1^.ST03_552_B70_0.BitInToCheck} *)
	.ST03_552_Y70_1.CoilA AT %QX249.0 : BOOL;	(*  ~ {LinkedWith:TIID^Gerät 2 (EtherCAT)^946_A3 (EP2338-0001)^Channel 10^.ST03_552_Y70_1.CoilA} *)
	.ST03_552_Y70_1.CoilB AT %QX249.1 : BOOL;
	.ST03_552_Y70_2.CoilA AT %QX249.2 : BOOL;	(*  ~ {LinkedWith:TIID^Gerät 2 (EtherCAT)^946_A3 (EP2338-0001)^Channel 11^.ST03_552_Y70_2.CoilA} *)
	.ST03_552_Y70_2.CoilB AT %QX249.3 : BOOL;
	.ST03_556_B69_0.BitInToCheck AT %IX1408.3 : BOOL;
	.ST03_556_B69_1.ValveSensor AT %IX1408.4 : BOOL;
	.ST03_556_B69_2.ValveSensor AT %IX1408.5 : BOOL;
	.ST03_556_B69_3.ValveSensor AT %IX1408.6 : BOOL;
	.ST03_556_B69_4.ValveSensor AT %IX1408.7 : BOOL;
	.ST03_556_B69_5.BitInToCheck AT %IX1476.0 : BOOL;
	.ST03_556_B69_6.BitInToCheck AT %IX1409.0 : BOOL;
	.ST03_556_B69_7.BitInToCheck AT %IX1409.1 : BOOL;
	.ST03_557_Y70_1.CoilA AT %QX252.1 : BOOL;
	.ST03_557_Y70_1.CoilB AT %QX252.2 : BOOL;
	.ST03_557_Y70_2.CoilA AT %QX252.3 : BOOL;
	.ST03_557_Y70_2.CoilB AT %QX252.4 : BOOL;
	.ST03_562_B69_0.BitInToCheck AT %IX1409.2 : BOOL;
	.ST03_562_B69_1.ValveSensor AT %IX1409.3 : BOOL;
	.ST03_562_B69_2.ValveSensor AT %IX1409.4 : BOOL;
	.ST03_562_B69_3.ValveSensor AT %IX1409.5 : BOOL;
	.ST03_562_B69_4.ValveSensor AT %IX1409.6 : BOOL;
	.ST03_562_B69_6.BitInToCheck AT %IX1409.7 : BOOL;
	.ST03_562_B67_7.BitInToCheck AT %IX1410.0 : BOOL;
	.ST03_563_B70_0.BitInToCheck AT %IX1410.1 : BOOL;
	.ST03_563_B70_1.ValveSensor AT %IX1410.2 : BOOL;
	.ST03_563_B70_2.ValveSensor AT %IX1410.3 : BOOL;
	.ST03_563_B70_3.ValveSensor AT %IX1410.4 : BOOL;
	.ST03_563_B70_4.ValveSensor AT %IX1410.5 : BOOL;
	.ST03_563_B70_6.BitInToCheck AT %IX1410.6 : BOOL;
	.ST03_563_B70_7.BitInToCheck AT %IX1410.7 : BOOL;
	.ST03_564_Y71_0.CoilA AT %QX252.5 : BOOL;
	.ST03_564_Y71_0.CoilB AT %QX252.6 : BOOL;
	.ST03_564_Y71_1.CoilA AT %QX252.7 : BOOL;
	.ST03_564_Y71_1.CoilB AT %QX253.0 : BOOL;
	.ST03_564_Y71_2.CoilA AT %QX253.1 : BOOL;
	.ST03_564_Y71_2.CoilB AT %QX253.2 : BOOL;
	.ST03_564_Y71_3.CoilA AT %QX253.3 : BOOL;
	.ST03_564_Y71_3.CoilB AT %QX253.4 : BOOL;
	.ST03_564_Y71_4.CoilA AT %QX253.5 : BOOL;
	.ST03_564_Y71_4.CoilB AT %QX253.6 : BOOL;
	.ST03_564_Y71_5.CoilA AT %QX253.7 : BOOL;
	.ST03_564_Y71_5.CoilB AT %QX254.0 : BOOL;
	.ST03_565_B72_0.BitInToCheck AT %IX1411.0 : BOOL;
	.ST03_565_B72_1.BitInToCheck AT %IX1411.1 : BOOL;
	.ST03_565_B72_2.ValveSensor AT %IX1411.2 : BOOL;
	.ST03_565_B72_3.ValveSensor AT %IX1411.3 : BOOL;
	.ST03_565_B72_4.ValveSensor AT %IX1411.4 : BOOL;
	.ST03_565_B72_5.ValveSensor AT %IX1411.5 : BOOL;
	.ST03_565_B72_6.ValveSensor AT %IX1411.6 : BOOL;
	.ST03_565_B72_7.ValveSensor AT %IX1411.7 : BOOL;
	.ST03_571_B69_0.BitInToCheck AT %IX1440.1 : BOOL;
	.ST03_571_B69_1.BitInToCheck AT %IX1440.2 : BOOL;
	.ST03_571_B69_2.ValveSensor AT %IX1440.3 : BOOL;
	.ST03_571_B69_3.ValveSensor AT %IX1440.4 : BOOL;
	.ST03_571_B69_4.ValveSensor AT %IX1440.5 : BOOL;
	.ST03_571_B69_5.ValveSensor AT %IX1440.6 : BOOL;
	.ST03_571_B69_6.BitInToCheck AT %IX1440.7 : BOOL;
	.ST03_571_B69_7.BitInToCheck AT %IX1441.0 : BOOL;
	.ST03_572_Y70_0.CoilA AT %QX272.0 : BOOL;
	.ST03_572_Y70_0.CoilB AT %QX272.1 : BOOL;
	.ST03_572_Y70_1.CoilA AT %QX272.2 : BOOL;
	.ST03_572_Y70_1.CoilB AT %QX272.3 : BOOL;
	.ST08_412_B58_5_35pol.BitInToCheck AT %IX1304.0 : BOOL;	(*  ~ {LinkedWith:TIID^Gerät 2 (EtherCAT)^888_A1 (EP1816-0008)^DIG Inputs Channel 1^.ST08_412_B58_5.BitInToCheck} *)
	.ST08_412_B58_6_35pol.BitInToCheck AT %IX1304.1 : BOOL;	(*  ~ {LinkedWith:TIID^Gerät 2 (EtherCAT)^888_A1 (EP1816-0008)^DIG Inputs Channel 1^.ST08_412_B58_6.BitInToCheck} *)
	.ST08_180_M1.e_Position AT %IB1264 : UDINT;
	.ST08_180_M1.e_Statusword AT %IB1268 : UINT;
	.ST08_180_M1.e_Velocity AT %IB1270 : DINT;
	.ST08_180_M1.e_Torque AT %IB1332 : INT;
	.ST08_180_M1.e_Following_Error AT %IB1274 : DINT;
	.ST08_180_M1.e_Toggle AT %IX1278.0 : BOOL;
	.ST08_180_M1.e_State AT %IB1384 : UINT;
	.ST08_180_M1.a_Controlword AT %QB152 : UINT;
	.ST08_180_M1.a_Target_Velocity AT %QB154 : DINT;
	.ST08_180_M1.a_Target_Position AT %QB158 : UDINT;
	.ST08_185_M1.e_Position AT %IB1279 : UDINT;
	.ST08_185_M1.e_Statusword AT %IB1283 : UINT;
	.ST08_185_M1.e_Velocity AT %IB1285 : DINT;
	.ST08_185_M1.e_Torque AT %IB1334 : INT;
	.ST08_185_M1.e_Following_Error AT %IB1289 : DINT;
	.ST08_185_M1.e_Toggle AT %IX1293.0 : BOOL;
	.ST08_185_M1.e_State AT %IB1386 : UINT;
	.ST08_185_M1.a_Controlword AT %QB162 : UINT;
	.ST08_185_M1.a_Target_Velocity AT %QB164 : DINT;
	.ST08_185_M1.a_Target_Position AT %QB168 : UDINT;
	.ST08_190_M1.e_Position AT %IB1444 : UDINT;
	.ST08_190_M1.e_Statusword AT %IB1448 : UINT;
	.ST08_190_M1.e_Velocity AT %IB1450 : DINT;
	.ST08_190_M1.e_Torque AT %IB1454 : INT;
	.ST08_190_M1.e_Following_Error AT %IB1456 : DINT;
	.ST08_190_M1.e_Toggle AT %IX1460.0 : BOOL;
	.ST08_190_M1.e_State AT %IB1461 : UINT;
	.ST08_190_M1.a_Controlword AT %QB276 : UINT;
	.ST08_190_M1.a_Target_Velocity AT %QB278 : DINT;
	.ST08_190_M1.a_Target_Position AT %QB282 : UDINT;
END_VAR

(* Data type in zLibrary/CSV_Handling *)
TYPE CSV_Config :
STRUCT
	ColName				:STRING(30);
	ColDataType			:INT;
	ColSourceAdr		:DWORD;
	ColSourceSize		:DWORD;

END_STRUCT
END_TYPE

(* Data type in zLibrary/CSV_Handling *)
TYPE DataTypeDef :
STRUCT

	iBOOL		:INT:=1;
	iBYTE		:INT:=2;
	iWORD		:INT:=3;
	iDWORD		:INT:=4;
	iSINT		:INT:=5;
	iUSINT		:INT:=6;
	iINT		:INT:=7;
	iUINT		:INT:=8;
	iDINT		:INT:=9;
	iUDINT		:INT:=10;
	iREAL		:INT:=11;
	iLREAL		:INT:=12;
	iSTRING		:INT:=13;
	iTIME		:INT:=14;
	iTOD		:INT:=15;
	iDATE		:INT:=16;
	iDT			:INT:=17;

END_STRUCT
END_TYPE

(* Data type in System/Error_and_Message *)
TYPE eMsgDataLineType :
	(
	MsgDataTypeNone			:=	0,
	MsgDataTypeBool			:=	1,
	MsgDataTypeDint			:=	2,
	MsgDataTypeReal			:=	3,
	MsgDataTypeString		:=	4
	);
END_TYPE

(* Data type in zLibrary/AnaIn *)
TYPE enum_Drehrichtung :
	(
	RUECKWAERTS := -1,
	STEHT := 0,
	VORWAERTS := 1
	);
END_TYPE

(* Data type in System/LanguageHandler *)
TYPE enum_Lng :
(
	DE 			:=	0,
	EN			:=	1,
	CZ			:=	2

);
END_TYPE

(* Data type in EPT Lib/Achsen/EL72x1 *)
TYPE enum_ModeOfOperation :
	(
	CSP			:=	8,	(*cyclic synchronous position*)
	CSV			:=	9,	(*cyclic synchronous velocity*)
	CST			:=	10,	(*cyclic synchronous torque*)
	CSTCA		:=	11	(*cyclic synchronous torque with commutation angle*)
	);
END_TYPE

(* Data type in EPT Lib/Hydra *)
TYPE enum_StatusId :
	(

		(*
		M_S = Maschinenstörung,
		W_S = Werkzeugstörung,
		P_S = Peripheriestörung,
		AOI_S = Kamerastörung,
		M_W = Maschinenwartung,
		W_W = Werkzeugwartung,
		A_U = Ablaufunterbrechung
		*)


		_PRODUKTION := 1,
		_Nachtabschaltung_STOP := 199,
		_S_Quittiert := 290,
		_A_U_Steuerung_Aus := 299,
		_A_U_Auftrag_voll := 300,
		_M_S_Haube_Einzug := 301,
		_A_U_Trennstelle := 303,
		_A_U_Spule_voll := 304,
		_M_S_Haubenschaltleiste := 305,
		_M_S_Haube_Bandauslauf := 306,
		_M_S_Klappe_hinten := 307,
		_M_S_Klappe_links := 308,
		_M_S_Klappe_rechts := 309,
		_M_S_Klappe_vorne := 310,
		_M_S_Temp_Schaltschrank := 311,
		_M_S_Temp_Haubenmotor := 312,
		_M_S_Temp_Haubenluefter := 313,
		_M_S_Bandoeler_Fuellstand := 314,
		_M_S_Bandoeler := 315,
		_M_W_Pressenkopf := 316,
		_M_W_Zahnriemen := 317,
		_M_W_Wartungseinheit := 318,
		_M_W_Bandeinzug := 319,
		_M_W_Werkzeug := 320,
		_M_S_Drehgeber := 321,
		_M_S_Hauptantriebsmotor := 322,
		_M_S_Abfallbehaelter := 323,
		_W_S_Bandaufgestellt := 325,
		_W_S_Parallelschnitt := 326,
		_W_S_Gesamtschnitt_o := 327,
		_W_S_Gesamtschnitt_u := 328,
		_W_S_Dyn_Schnittueberw_eins := 329,
		_W_S_Dyn_Schnittueberw_zwei := 331,
		_W_S_Faengerueberw_eins := 332,
		_W_S_Faengerueberw_zwei := 333,
		_W_S_Faengerueberw_drei := 334,
		_W_S_Faengerueberw_vier := 335,
		_W_S_Position_Wkz := 336,
		_W_S_Pfostenabfrage := 337,
		_W_S_Tcom_eins := 338,
		_W_S_Tcom_zwei := 339,
		_W_S_Bandschneideueberwachung := 340,
		_W_S_Pinabstanzueberwachung := 341,
		_AOI_S_Kamera :=343,
		_P_S_Aufhaspel := 350,
		_P_S_Abhaspel := 351,
		_M_S_Not_Halt := 352,
		_M_S_Auffahrsicherung := 353,
		_Trennstelle := 809,
		_Maschine_STOP :=843,
		_Peripherie_STOP := 844,
		_Stoerung_Lasertriangulation := 870,
		_Stoerung_Bsh_Zellen := 871,
		_Maschinenstoerung := 884,
		_Peripheriestoerung := 885,
		_WERKZEUGSTOERUNG := 886,
		 _Kamerastoerung := 887,
		_HV_Stoerung := 888,
		_Schichtfrei := 999

);

END_TYPE

(* Data type in EPT Lib/Allgemeine Kontrollstrukturen Objekte *)
TYPE enum_step_nr :
	(
	INIT_OBJ := 0,
	INIT := 10,
	BEREIT := 100,
	HALT := 970,
	STOP := 980,
	FEHLER := 1000,
	INAKTIV:=2010
	);
END_TYPE

(* Data type in System/Error_and_Message *)
TYPE ErrorStruct :
STRUCT
	No							: DINT;
	DateTime					: DT;
	Text						: STRING(255);
	Typ							: DINT; (* 0=FatalError , 1=Warning, 2=OperatorInfo *)
	Station						: DINT;
	Prio						: DINT; (*1=heighest, .. , 4=lowest*)
	QuitAddr					: DWORD;
	LineColor					: DINT;
(*	Instance					: STRING;*)
END_STRUCT
END_TYPE

(* Data type in zLibrary/Sensopart *)
TYPE eSensopartCommands:
	(
	Sensopart_Connect			:=10,
	Sensopart_Trigger			:=20
	);
END_TYPE

(* Data type in sStation/sMachineParameter/Service *)
TYPE eService_Type :
	(
	BETRIEBSSTUNDEN			:=	0,
	STUNDEN			:=	1,
	TAGE				:=	2,
	COUNTER			:=	3
	);
END_TYPE

(* Data type in System/SystemSettings *)
TYPE eTargetSystem :
	(
	TARGETSYSTEM_CE					:=  1,   (* TaragetSystem with Winwows CE *)
	TARGETSYSTEM_XPP				:=  2,   (* TaragetSystem with Winwows XP Pro SP 3 *)
	TARGETSYSTEM_LOCAL_C		:=  3,   (* TaragetSystem on Developmant System - Path Mapped to Drive C *)
	TARGETSYSTEM_LOCAL_D		:=  4    (* TaragetSystem on Developmant System - Path Mapped to Drive D *)
	);
END_TYPE

(* Data type in sStation *)
TYPE PartState :
(
	PART_NO			:= 0, (*no Part available*)
	PART_OK			:= 1, (*Part processed with OK-Result*)
	PART_NOK		:= 2, (*Part processed with NOK-Result*)
	PART_NEW		:= 4,  (*new Part (picked up from Feeder, and not yet processed) *)
	PART_CAM		:= 5	(*Part muss zur Kamera*)
);
END_TYPE

(* Data type in zLibrary/AnaIn *)
TYPE sAnaInInit :
STRUCT
	InstName				:STRING(20);	(* Name of instance  *)
	Description				:STRING(32);	(* Description  *)
	BitInName				:STRING(25);	(* Name of bit input *)
	ScalingSensorValueMin	:INT;			(* min Scaling Value from Sensor *)
	ScalingSensorValueMax	:INT;			(* max Scaling Value from Sensor *)
	ScalingOutputValueMin	:REAL;			(* min Scaling Value on Output *)
	ScalingOutputValueMax	:REAL;			(* max Scaling Value on Output *)

END_STRUCT
END_TYPE

(* Data type in zLibrary/AnaIn *)
TYPE sAnaInVisu :
STRUCT
	InstName			:STRING(20);	(* Name of instance  *)
	Description			:STRING(32);	(* Description  *)
	BitInName			:STRING(25);	(* Name of bit input  *)

(* Outputvariables *)
	State				:DINT;			(* State of the outinput check *)
	AnaInValue			:REAL;
	HomePosition		:BOOL;			(* Object in home position  *)
	ErrorString			:STRING(40);	(* string shows missing signal *)
	ErrorPresent			: BOOL;
END_STRUCT
END_TYPE

(* Data type in System/VisuInterface *)
TYPE sButtonVisu :
STRUCT
		Visible				: BOOL;
		Enable				: BOOL;
		Pressed				: BOOL;
		Text				: STRING;
		TextColor			: DINT;
		BackgroundColor	: DINT ;
		Tasten				: BOOL;
END_STRUCT
END_TYPE

(* Data type in System/VisuInterface *)
TYPE sButtonVisu_Tree :
STRUCT
	unsichtbar				: BOOL;
	deaktivieren				: BOOL;
	tasten					: BOOL;
	Textfarbe				: DINT;
	innenFarbe				: DINT;
	Text					: STRING(50);
	Zoom					: STRING(50);
END_STRUCT
END_TYPE

(* Data type in System/VisuInterface *)
TYPE sButtonVisuBmp :
STRUCT
	unsichtbar			: BOOL;
	deaktivieren		: BOOL;
	tasten				: BOOL;
	Text				: STRING(30);
	Textfarbe			: DINT;
	innenFarbe			: DINT;
	BmpPath				: STRING(255);
END_STRUCT
END_TYPE

(* Data type in System/VisuInterface *)
TYPE sColorCode :
STRUCT
	black				:    DINT  :=  16#000000;
	maroon   			:    DINT  :=  16#000080;
	green  				:    DINT  :=  16#008000;
	olive    				:    DINT  :=  16#008080;
	navy    				:    DINT  :=  16#800000;
	purple    			:    DINT  :=  16#800080;
	teal    				:    DINT  :=  16#808000;
	grey    				:    DINT  :=  16#808080;
	silver    			:    DINT  :=  16#C0C0C0;
	red    				:    DINT  :=  16#0000FF;
	lime    				:    DINT  :=  16#00FF00;
	yellow    			:    DINT  :=  16#00FFFF;
	blue    				:    DINT  :=  16#FF0000;
	fuchsia    			:    DINT  :=  16#FF00FF;
	aqua    			:    DINT  :=  16#FFFF00;
	white    			:    DINT  :=  16#FFFFFF;
	aliceblue    		:    DINT  :=  16#FFF8F0;
	antiquewhite   	:    DINT  :=  16#D7EBFA;
	aquamarine    :    DINT  :=  16#D4FF7F;
	azure    			:    DINT  :=  16#FFFFF0;
	beige    			:    DINT  :=  16#DCF5F5;
	blueviolet    	:    DINT  :=  16#E22B8A;
	brown    			:    DINT  :=  16#2A2AA5;
	burlywood    	:    DINT  :=  16#87B8DE;
	cadetblue    :    DINT  :=  16#A09E5F;
	chartreuse    :    DINT  :=  16#00FF7F;
	chocolate    :    DINT  :=  16#1E69D2;
	coral    :    DINT  :=  16#507FFF;
	cornflowerblue    :    DINT  :=  16#ED9564;
	cornsilk    :    DINT  :=  16#DCF8FF;
	crimson    :    DINT  :=  16#3C14DC;
	darkblue    :    DINT  :=  16#8B0000;
	darkcyan    :    DINT  :=  16#8B8B00;
	darkgoldenrod    :    DINT  :=  16#0B86B8;
	darkgrey    :    DINT  :=  16#A9A9A9;
	darkgreen    :    DINT  :=  16#006400;
	darkkhaki    :    DINT  :=  16#6BB7BD;
	darkmagenta    :    DINT  :=  16#8B008B;
	darkolivegreen    :    DINT  :=  16#2F6B55;
	darkorange    :    DINT  :=  16#008CFF;
	darkorchid    :    DINT  :=  16#CC3299;
	darkred    :    DINT  :=  16#00008B;
	darksalmon    :    DINT  :=  16#7A96E9;
	darkseagreen    :    DINT  :=  16#8FBC8F;
	darkslateblue    :    DINT  :=  16#8B3D48;
	darkslategrey    :    DINT  :=  16#4F4F2F;
	darkturquoise    :    DINT  :=  16#D1CE00;
	darkviolet    :    DINT  :=  16#D30094;
	deeppink    :    DINT  :=  16#9314FF;
	deepskyblue    :    DINT  :=  16#FFBF00;
	dimgrey    :    DINT  :=  16#696969;
	dodgerblue    :    DINT  :=  16#FF901E;
	firebrick    :    DINT  :=  16#2222B2;
	floralwhite    :    DINT  :=  16#F0FAFF;
	forestgreen    :    DINT  :=  16#228B22;
	gainsboro    :    DINT  :=  16#DCDCDC;
	ghostwhite    :    DINT  :=  16#FFF8F8;
	gold    :    DINT  :=  16#00D7FF;
	goldenrod    :    DINT  :=  16#20A5DA;
	greenyellow    :    DINT  :=  16#2FFFAD;
	honeydew    :    DINT  :=  16#F0FFF0;
	hotpink    :    DINT  :=  16#B469FF;
	indianred    :    DINT  :=  16#5C5CCD;
	indigo    :    DINT  :=  16#82004B;
	ivory    :    DINT  :=  16#F0FFFF;
	khaki    :    DINT  :=  16#8CE6F0;
	lavender    :    DINT  :=  16#FAE6E6;
	lavenderblush    :    DINT  :=  16#F5F0FF;
	lawngreen    :    DINT  :=  16#00FC7C;
	lemonchiffon    :    DINT  :=  16#CDFAFF;
	lightblue    :    DINT  :=  16#E6D8AD;
	lightcoral    :    DINT  :=  16#8080F0;
	lightcyan    :    DINT  :=  16#FFFFE0;
	lightgoldenrodyellow    :    DINT  :=  16#D2FAFA;
	lightgreen    :    DINT  :=  16#90EE90;
	lightgrey    :    DINT  :=  16#D3D3D3;
	lightpink    :    DINT  :=  16#C1B6FF;
	lightsalmon    :    DINT  :=  16#7AA0FF;
	lightseagreen    :    DINT  :=  16#AAB220;
	lightskyblue    :    DINT  :=  16#FACE87;
	lightslategrey    :    DINT  :=  16#998877;
	lightsteelblue    :    DINT  :=  16#DEC4B0;
	lightyellow    :    DINT  :=  16#E0FFFF;
	limegreen    :    DINT  :=  16#32CD32;
	linen    :    DINT  :=  16#E6F0FA;
	mediumaquamarine    :    DINT  :=  16#AACD66;
	mediumblue    :    DINT  :=  16#CD0000;
	mediumorchid    :    DINT  :=  16#D355BA;
	mediumpurple    :    DINT  :=  16#D7093;
	mediumseagreen    :    DINT  :=  16#71B33C;
	mediumslateblue    :    DINT  :=  16#EE687B;
	mediumspringgreen    :    DINT  :=  16#9AFA00;
	mediumturquoise    :    DINT  :=  16#CCD148;
	mediumvioletred    :    DINT  :=  16#8515C7;
	midnightblue    :    DINT  :=  16#701919;
	mintcream    :    DINT  :=  16#FAFFF5;
	mistyrose    :    DINT  :=  16#E1E4FF;
	moccasin    :    DINT  :=  16#B5E4FF;
	navajowhite    :    DINT  :=  16#ADDEFF;
	oldlace    :    DINT  :=  16#E6F5FD;
	olivedrab    :    DINT  :=  16#238E6B;
	orange    :    DINT  :=  16#00A5FF;
	orangered    :    DINT  :=  16#0045FF;
	orchid    :    DINT  :=  16#D670DA;
	palegoldenrod    :    DINT  :=  16#AAE8EE;
	palegreen    :    DINT  :=  16#98FB98;
	paleturquoise    :    DINT  :=  16#EEEEAF;
	palevioletred    :    DINT  :=  16#9370DB;
	papayawhip    :    DINT  :=  16#D5EFFF;
	peachpuff    :    DINT  :=  16#B9DAFF;
	peru    :    DINT  :=  16#3F85CD;
	pink    :    DINT  :=  16#CBC0FF;
	plum    :    DINT  :=  16#DDA0DD;
	powderblue    :    DINT  :=  16#E6E0B0;
	rosybrown    :    DINT  :=  16#8F8FBC;
	royalblue    :    DINT  :=  16#E16941;
	saddlebrown    :    DINT  :=  16#13458B;
	salmon    :    DINT  :=  16#7280FA;
	sandybrown    :    DINT  :=  16#60A4F4;
	seagreen    :    DINT  :=  16#578B2E;
	seashell    :    DINT  :=  16#EEF5FF;
	sienna    :    DINT  :=  16#2D52A0;
	skyblue    :    DINT  :=  16#EBCE87;
	slateblue    :    DINT  :=  16#CD5A6A;
	slategrey    :    DINT  :=  16#908070;
	snow    :    DINT  :=  16#FAFAFF;
	springgreen    :    DINT  :=  16#7FFF00;
	steelblue    :    DINT  :=  16#B48246;
	thistle    :    DINT  :=  16#D8BFD8;
	tomato    :    DINT  :=  16#4763FF;
	turquoise    :    DINT  :=  16#D0E040;
	violet    :    DINT  :=  16#EE82EE;
	wheat    :    DINT  :=  16#B3DEF5;
	whitesmoke    :    DINT  :=  16#F5F5F5;
	yellowgreen    :    DINT  :=  16#32CD9A;
 	control    :    DINT  :=  16#D3D3D3;
(*	control    :    DINT  :=  16#D8E9EC;*)



END_STRUCT
END_TYPE

(* Data type in EPT Lib/sDatensatz/sTypeDaten *)
TYPE sData_b :
STRUCT

	Description					: STRING(50); 	(* Beschreibung *)
	b								: BOOL; 		(* Wert *)

END_STRUCT
END_TYPE

(* Data type in EPT Lib/sDatensatz/sTypeDaten *)
TYPE sData_byte :
STRUCT

	Description					: STRING(50); 	(* Beschreibung *)
	BYT								: BYTE; 			(* Wert *)
	Unit				   			: STRING(20);	(* Einheit *)

END_STRUCT
END_TYPE

(* Data type in EPT Lib/sDatensatz/sTypeDaten *)
TYPE sData_i16 :
STRUCT

	Description					: STRING(50); 	(* Beschreibung *)
	i16								: INT; 			(* Wert *)
	Unit				   			: STRING(20);	(* Einheit *)

END_STRUCT
END_TYPE

(* Data type in EPT Lib/sDatensatz/sTypeDaten *)
TYPE sData_i32 :
STRUCT

	Description		: STRING(50); 	(* Beschreibung *)
	i32					: DINT; 		(* Wert *)
	Unit				: STRING(20);	(* Einheit *)

END_STRUCT
END_TYPE

(* Data type in EPT Lib/sDatensatz/sTypeDaten *)
TYPE sData_lr :
STRUCT

	Description		: STRING(50); 	(* Beschreibung *)
	lr					: LREAL; 			(* Wert *)
	Unit		   		: STRING(20);	 	(* Einheit *)

END_STRUCT
END_TYPE

(* Data type in EPT Lib/sDatensatz/sTypeDaten *)
TYPE sData_Str :
STRUCT

	Description				: STRING(50); 	(* Beschreibung *)
	str							: STRING(50); 	(* Text *)

END_STRUCT
END_TYPE

(* Data type in EPT Lib/sDatensatz/sTypeDaten *)
TYPE sData_ui32 :
STRUCT

	Description			: STRING(50); 	(* Beschreibung *)
	i32						: UDINT; 		(* Wert *)
	Unit					: STRING(20);	(* Einheit *)

END_STRUCT
END_TYPE

(* Data type in zLibrary/DigIn *)
TYPE sDigInInit :
STRUCT
	InstName			: STRING(25);		(* Name of instance  *)
	Description			: STRING(50);		(* Description  *)
	BitInName			: STRING(25);		(* Name of bit input *)
	HomePosSignal		: DINT;				(* home-position is definded if : 0: Signal=Low, 1: Signal=High, 2: always  *)
	MaxTime				: DINT; 			(* number in ms cycles to Timeout *)
	EnableInEveryMode	: BOOL;				(* Object can be Controlled in every Mode *)

	IputOnDelayTime		: DINT;				(* number in ms for On - Delay SignalInDelayed *)
	IputOffDelayTime	: DINT;				(* number in ms for On - Delay SignalInDelayed *)

END_STRUCT
END_TYPE

(* Data type in zLibrary/DigIn *)
TYPE sDigInVisu :
STRUCT
	InstName				: STRING(25);		(* string shows instance name *)
	Description				: STRING(50);		(* Description        *)
	BitInName				: STRING(25);		(* Name of bit input  *)

(* Inputvariables *)
	BtnReset				: sButtonVisu;		(* Manage button *)

(* Outputvariables *)
	State					: StateObject;			(* State of the outinput check *)
	HomePosition			: BOOL;					(* Object in home position  *)
	ErrorString				: STRING(40);			(* string shows missing signal *)
	ErrorPresent			: BOOL;

(* Internal variables *)
	BitInToCheck			: BOOL;					(* Bit input signal  *)
	ProcessTime				: DINT;					(* Counts the time in ms						*)
	BtnResetVisible			: BOOL;					(* Switch for reset the input check *)

END_STRUCT
END_TYPE

(* Data type in zLibrary/DigOutIn *)
TYPE sDigOutInHome :
(
	HOME_LOW			:=0,
	HOME_HIGH 			:=1,
	HOME_NOT_DEFINED 	:=2

);
END_TYPE

(* Data type in zLibrary/DigOutIn *)
TYPE sDigOutInInit :
STRUCT
	InstName				: STRING(25);	(* Name of instance  *)
	Description				: STRING(50);	(* Description  *)

	BitOutName				: STRING(25);	(* Name of bit output*)
	BitInName				: STRING(25);	(* Name of bit input *)
	HomePosSignal			: DINT;			(* home-position is definded if :
															 	0: Signal=Low, 1: Signal=High, 2: always  *)
	HomePosOutput			: DINT;			(* home-position is definded if :
															 	0: Output=Low, 1: Output=High, 2: always  *)
	MaxTime					: DINT; 			(* number in ms cycles to Timeout *)
	EnableInEveryMode		: BOOL;			(* Object can be Controlled in every Mode *)
	EnableVisuInEveryMode	: BOOL;			(* Object can be Controlled from Visu in every Mode *)

END_STRUCT
END_TYPE

(* Data type in zLibrary/DigOutIn *)
TYPE sDigOutInVisu :
STRUCT
	InstName				:STRING(25);	(* string shows instance name *)
	Description				:STRING(50);	(* Description        *)
	BitOutName				:STRING(25);	(* Name of bit output *)
	BitInName				:STRING(25);	(* Name of bit input *)

(* Inputvariables *)
	BtnOutput				:sButtonVisu;	(* Manage button *)

(* Outputvariables *)
	State					:StateObject;	(* State of the outinput check *)
	OutputAvailable			:BOOL;			(* Output available *)
	InputAvailable			:BOOL;			(* Input available 	*)
	HomePosition			:BOOL;			(* Object in home position  *)
	ErrorString				:STRING(40);	(* string shows missing signal *)
	ErrorPresent			: BOOL;

(* Internal variables *)
	BitOutToSet				:BOOL;			(* Bit output signal *)
	BitInToCheck			:BOOL;			(* Bit input signal  *)
	ProcessTime				:DINT;			(* Counts the time in ms *)
	BtnResetVisible			:BOOL;			(* Switch for reset the input check *)
END_STRUCT
END_TYPE

(* Data type in zLibrary/AnaIn *)
TYPE sEncoderInit :
STRUCT
	InstName				:STRING(20);	(* Name of instance  *)
	Description				:STRING(32);	(* Description  *)
	BitInName				:STRING(25);	(* Name of bit input *)

	lr_LaengeProRpm			:LREAL;			(* mm *)
	i_InkProRpm				:UDINT		:=1440;		(*360 * 4*)	(* Inkremente pro Umdehung *)
END_STRUCT
END_TYPE

(* Data type in zLibrary/AnaIn *)
TYPE sEncoderVisu :
STRUCT
	InstName			:STRING(20);	(* Name of instance  *)
	Description			:STRING(32);	(* Description  *)
	BitInName			:STRING(25);	(* Name of bit input  *)

	Reset				:BOOL;

(* Outputvariables *)
	State				:DINT;			(* State of the outinput check *)
	ErrorString			:STRING(40);	(* string shows missing signal *)
	ErrorPresent			: BOOL;
	Drehrichtung		:enum_Drehrichtung;
	rpmValue			:LREAL;			(* rpm *)
	posValue			:LREAL;			(* mm *)
END_STRUCT
END_TYPE

(* Data type in zLibrary/EsponRobot *)
TYPE sEpsonRobotInit :
STRUCT
(* Structure for initialising a valve *)
	BitName				: STRING(20);	(* Name of bit *)
	InstName			: STRING(20);	(* Instance name of the object *)
	Description			: STRING(50);	(* Description of instance *)

	MaxTime				: DINT; 			(* number of 100ms cycles to Timeout *)
	TcpIPSocket			: DINT; 			(* Socket No of TCP-IP Connection *)
	TcpIPAdress			: STRING(16); 	(* IP-Adress of TCP-IP Connection *)
	WithToolHandling	: BOOL;
	ToolMaxTime			: DINT;

END_STRUCT
END_TYPE

(* Data type in zLibrary/EsponRobot *)
TYPE sEpsonRobotRecvData :
STRUCT
	Alive			: DINT;
	TelNo			: DINT;
	PosNo			: DINT;
	PosX			: REAL;
	PosY			: REAL;
	PosZ			: REAL;
	ApplPara		: ARRAY[0..7] OF	REAL;
	ErrorCode		: DINT;

END_STRUCT
END_TYPE

(* Data type in zLibrary/EsponRobot *)
TYPE sEpsonRobotSendData :
STRUCT
	Alive			:	DINT;
	TelNo			:	DINT;
	PosNo			:	DINT;
	Override	:	DINT;
	Vel				:	DINT;
	Acc				:	DINT;
	OffsetX			:	REAL;
	OffsetY			:	REAL;
	OffsetZ			:	REAL;
	ApplPara	:	ARRAY[0..7] OF	REAL;

END_STRUCT
END_TYPE

(* Data type in zLibrary/EsponRobot *)
TYPE sEpsonRobotToolSettings :
STRUCT
(* Structure for initialising robot tool *)
	NameCoilA			: STRING(20);
	NameCoilB			: STRING(20);
	NameInitSensor		: STRING(20);
	NameWorkSensor	: STRING(20);
	NameBtnToolOn		: STRING(30);
	NameBtnToolOff		: STRING(30);
END_STRUCT
END_TYPE

(* Data type in zLibrary/EsponRobot *)
TYPE sEpsonRobotVisu :
STRUCT
(* Structure for Handshake to display a Epson Robot *)
(*--------------------------------------------------------------*)
(* sInit-Datas *)
	BitName					: STRING(20);	(* Name of bit *)
	InstName					: STRING(20);	(* Instance name of the object *)
	Description					: STRING(50);	(* Description of instance *)
	TcpIpAdress				: STRING(15);
	SocketState 				: STRING(20);

(* sRobotToolSetting-Datas *)
	WithToolHandling			: BOOL;
	NameCoilA					: STRING(20);
	NameCoilB					: STRING(20);
	NameInitSensor				: STRING(20);
	NameWorkSensor			: STRING(20);

(* Outputvariables*)
	State						: StateObject;	(* State of the valve*)
	HomePosition				: BOOL; 		(* valve in home-position*)
	ErrorString					: STRING(80);	(* string shows missing signal*)
	ErrorPresent					: BOOL;
	ActualPosition				: DINT;
	ActualArea					: DINT;
	ConnectionAlive				: BOOL;
	PosX						: REAL;
	PosY						: REAL;
	PosZ						: REAL;
	PosArray					: ARRAY[1..20] OF STRING(30);

(* From Visu to Object *)
	PosNo						: DINT;			(* Position No from Robot *)
	OffsetX						: REAL;			(* Offset X *)
	OffsetY						: REAL;			(* Offset Y *)
	OffsetZ						: REAL;			(* Offset Z *)
	ApplPara					: ARRAY[0..7] OF REAL; (* Machinespecific Values *)

(* Internal Variables*)
	ProcessTime				: DINT;			(* Counts the time in ms*)
	PosOffset					: DINT;

	BtnMove					: sButtonVisu;	(* Manage button *)
	BtnReset					: sButtonVisu;	(* Manage button *)
	BtnPrgStart					: sButtonVisu;	(* Manage button *)
	BtnPrgStop					: sButtonVisu;	(* Manage button *)
	BtnToolOn 					: sButtonVisu;	(* Manage button *)
	BtnToolOff					: sButtonVisu;	(* Manage button *)

(* Internal Variables used only in Visu *)
	ShowDetails					: BOOL;
	ShowPosArray				: BOOL;

(* EA's from Robot *)
	RemOutStart				: BOOL; 		(* For Moving to WorkPosition *)
	RemOutStop				: BOOL; 		(* For Moving to WorkPosition *)
	RemOutPause				: BOOL; 		(* For Moving to WorkPosition *)
	RemOutCont				: BOOL; 		(* For Moving to WorkPosition *)
	RemOutReset				: BOOL; 		(* For Moving to WorkPosition *)
	RemOutPowerOn			: BOOL; 		(* For Moving to WorkPosition *)
	RemOutPowerOff			: BOOL; 		(* For Moving to WorkPosition *)
	RemOutPowerHi				: BOOL; 		(* For Moving to WorkPosition *)
	RemOutSetToolOn			: BOOL; 		(* Anforderung Ausgang Robotertool EIN *)
	RemOutSetToolOff			: BOOL; 		(* Anforderung Ausgang Robotertool AUS *)

	RemInReady				: BOOL; 		(* For Moving to WorkPosition *)
	RemInRunning				: BOOL; 		(* For Moving to WorkPosition *)
	RemInPaused				: BOOL; 		(* For Moving to WorkPosition *)
	RemInError					: BOOL; 		(* For Moving to WorkPosition *)
	RemInEStopOn				: BOOL; 		(* For Moving to WorkPosition *)
	RemInSafeguardOn			: BOOL; 		(* For Moving to WorkPosition *)
	RemInSError				: BOOL; 		(* For Moving to WorkPosition *)
	RemInWarning				: BOOL; 		(* For Moving to WorkPosition *)

	RemInTcpIP_Wait			: BOOL; 		(* For Moving to WorkPosition *)
	RemInAreaBit1				: BOOL; 		(* For Moving to WorkPosition *)
	RemInAreaBit2				: BOOL; 		(* For Moving to WorkPosition *)
	RemInAreaBit4				: BOOL; 		(* For Moving to WorkPosition *)

	RemInToolCoilA				: BOOL;			(* Rückmeldung Tool CoilA/ Ausgang 1 ist ein *)
	RemInToolCoilB				: BOOL;			(* Rückmeldung Tool CoilB/ Ausgang 2 ist ein *)
	RemInToolInitSensor			: BOOL;			(* Tool Ruhesensor *)
	RemInToolWorkSensor		: BOOL;			(* Tool Ruhesensor *)

END_STRUCT
END_TYPE

(* Data type in System/Error_and_Message *)
TYPE sErrorHandlerVisu :
STRUCT
	Error								:	ARRAY[0..NO_OF_ERRORS] OF ErrorStruct;
	ScrollBarShow				:	BOOL;
	ScrollBarMax				:	DINT;
	ScrollBarPosition		:	DINT;
END_STRUCT
END_TYPE

(* Data type in sStation *)
TYPE SFCCurrent :
STRUCT
	SFCCurrentPOU		: STRING:=	'-';
	SFCCurrentStep		: STRING;
	SFCTime			: DINT;
	b_activ				: BOOL;
END_STRUCT
END_TYPE

(* Data type in sStation/sMachineParameter *)
TYPE sMachineParameterHandling :
STRUCT
(* ST01 *)
	Dummy:BOOL;
(* ST02 *)

(* ST03 *)

(* ST04 *)

(* ST05 *)
END_STRUCT
END_TYPE

(* Data type in sStation/sMachineParameter *)
TYPE sMachPara :
STRUCT
	sLastTDfile							: STRING;
	ShiftData							: sMP_ShiftHandler;
	ST00: sMachParaST00; (*Instancename is Filename in Typedata Folder*)
	ST02: sMachParaST02; (*Instancename is Filename in Typedata Folder*)
	ST03: sMachParaST03; (*Instancename is Filename in Typedata Folder*)
	ST08: sMachParaST08; (*Instancename is Filename in Typedata Folder*)
	Visu:	sMachineParameterHandling; (* Object Collection for Parameterhandling in Visu - e.g. Buttons - Called in System/VisuInterface/MachParaHandling  *)
END_STRUCT
END_TYPE

(* Data type in sStation/sMachineParameter/Service *)
TYPE sMachParaService :
STRUCT
	visu			: ARRAY[0..15] OF struct_visu_service;
	daten			: ARRAY[0..15] OF struct_daten_service;
	betriebssekundenzaehler	:UDINT;
END_STRUCT
END_TYPE

(* Data type in sStation/sMachineParameter *)
TYPE sMachParaST00 :
STRUCT
	Override					:	DINT :=10;
	OverrideForHoming	:	DINT :=5;
	MaxLogInTime				: DINT  := 0;
	Sprache    					: STRING(10);

	ActPartNo			: DINT; (*laufende Nr. für Laser-String*)

	IFMCameraActive			: BOOL := TRUE;
	IFMCameraActiveText		:STRING :='ON';

	Cam_NoOfErrors		: DINT := 1;

(* -----------------------------------------------------------------------------------------
		Sollwerte
  ----------------------------------------------------------------------------------------- *)

	PartsToProduce					: DINT;		(* Sollstückzahl *)
	PartsToProduceOffset		: DINT;		(* Korrenkturwert auf Sollstückzahl *)

 	PartsNokInSeriesAllowed : DINT := 0;		(* max. Fehler in Folge *)

	PartsNokPerSubset				: DINT :=0;		(* max. erlaubete n.i.O. Teileanzahl pro Untermenge *)
	PartsNokSubsetSize			: DINT :=100;		(* Untermengengröße *)

(* -----------------------------------------------------------------------------------------
		Istwerte
  ----------------------------------------------------------------------------------------- *)

	PartsInserted						: DINT;		(* Teile aufgesetzt in ST01 *)
	PartsNokTotal						: DINT;		(* Teile n.i.O. gesamt *)
	PartsOkTotal						: DINT;		(* Teile i.O. gesamt, eingesetzt in Blister/Tube *)
	PartsRemaining					: DINT;		(* Teile noch zu produzieren (PartsToProduce + PartsToProduceOffset + PartsNokTotal - PartsInserted) *)

	PartsNokTotalNoReset		: DINT;		(* Teile n.i.O. gesamt *)
	PartsOkTotalNoReset			: DINT;		(* Teile i.O. gesamt, eingesetzt in Blister/Tube *)

	LAN_no						: sData_i16:=(Description:='LAN_no', Unit:='no');
END_STRUCT
END_TYPE

(* Data type in sStation/sMachineParameter *)
TYPE sMachParaST02 :
STRUCT
	Override_Band				:	DINT :=10;

	RunTableEmpty 			: DINT := 5; (*Time in sec. *)
	IFMPos					: LREAL;
	IFMPosDummy			: LREAL;
	TableData				: ARRAY [1..NO_OF_NEST] OF sStationData;
	CamOn					: BOOL;
	CamNoOfErrors			: DINT := 1;
	CamNoOfErrorsPercent	: DINT := 1;
	DummyPruefung_93pol	: BOOL;
  	Dummy_test_Result  	: ARRAY [1..12] OF BOOL;
	NoOfDummys			: DINT := 6;
	SensopartIPAdress		: STRING(15);
	SensopartIPAdress2		: STRING(15);
	SensopartEthernet		: BOOL;

END_STRUCT
END_TYPE

(* Data type in sStation/sMachineParameter *)
TYPE sMachParaST03 :
STRUCT

	WpcInStackFilled		: BOOL;

	ActualPartsInPallet 		: DINT; (* Counter *)

	NoOfBlisterInStackerOut	: DINT; (* Counter *)

	ActualPartsOnBuffer 		: DINT; (* Counter *)

	ResetBuffer             : BOOL;
	(* Inputvariablen *)
	PartsInPallet	      	   : DINT; (* Max No Of Parts in Buffer *)

	NoOfTestParts				:	DINT;

	FrontCamOn			: BOOL;
	BackCamOn			: BOOL;
	CamNoOfErrors			: DINT := 1;
	CamNoOfErrorsPercent	: DINT := 1;

	RobotIPAdress			: STRING(15);
	BandMoveP				:BOOL;
	SGM_3621		: BOOL;

	BeltMotorCheckPartActive          : BOOL;

	RoboterColisionActivated	 :BOOL;

	CamOn					: ARRAY [1..2] OF BOOL;		(*Sensopart Kamera*)
	SensopartIPAdress		: ARRAY [1..2] OF STRING(15);

	CamOn_KYE				: BOOL;			(*Keyence Kamera*)
	CamNoOfErrors_KYE		: DINT := 1;
	CamNoOfErrorsPercent_KYE: DINT := 1;

END_STRUCT
END_TYPE

(* Data type in sStation/sMachineParameter *)
TYPE sMachParaST08 :
STRUCT
	NoOfBlisterInStackerOut			: DINT; (* Counter *)

	StapelMotor								: BOOL;
	PosOffsetAufstapeln	 			: st_Pos;
	PosOffsetAbstapeln	 			: st_Pos;
	Override_Aufstapeln				: DINT :=10;
	Override_Abstapeln				: DINT :=10;
	Traystapel_schieben 			: BOOL:=TRUE;
	Trayzufuhr_Verlaengerung		: BOOL:=TRUE;
	TrayAushebenMotor				: BOOL;
	PosOffsetTrayAusheben 			: st_Pos;
	Override_TrayAusheben			: DINT :=10;

END_STRUCT
END_TYPE

(* Data type in sStation/MainMenue *)
TYPE sMainMenue:
STRUCT
	BtnMainMenue					:sButtonVisu_Tree;
	BtnManual						:sButtonVisu_Tree;
	BtnManual_ST00_0				:sButtonVisu_Tree;	(*Allgemein*)
		BtnManual_ST00_1			:sButtonVisu_Tree;	(*Türen und Not-Halt*)
		BtnManual_ST00_2			:sButtonVisu_Tree;	(*Flügelkamera*)
	BtnManual_ST02_0				:sButtonVisu_Tree;	(*Rundtisch*)
	BtnManual_ST03_0				:sButtonVisu_Tree;	(*Roboter*)
			BtnManual_ST03_xx		:sButtonVisu_Tree;	(*Rüstsatz Seite1*)
			BtnManual_ST03_xx_2	:sButtonVisu_Tree;	(*Rüstsatz Seite2*)
	BtnManual_ST08_0				:sButtonVisu_Tree;
		BtnManual_ST08_1			:sButtonVisu_Tree;	(*Blisterzuführung*)
		BtnManual_ST08_2			:sButtonVisu_Tree;	(*Abstapeln*)
		BtnManual_ST08_3			:sButtonVisu_Tree;	(*Bandstrecke*)
		BtnManual_ST08_4			:sButtonVisu_Tree;	(*Aufstapeln*)


	BtnTD							:sButtonVisu_Tree;
	BtnTD01_Edit					:sButtonVisu_Tree;
	BtnTD02_Edit					:sButtonVisu_Tree;

	BtnMP_Main					:sButtonVisu_Tree;
	BtnMP_ST1						:sButtonVisu_Tree;
	BtnMP_ST2						:sButtonVisu_Tree;
	BtnMP_Date					:sButtonVisu_Tree;
	BtnMP_Service					:sButtonVisu_Tree;

	BtnSystem						:sButtonVisu_Tree;
		Btn_ErrorLog				:sButtonVisu_Tree;
		Btn_ErrorList				:sButtonVisu_Tree;
		Btn_Gst						:sButtonVisu_Tree;
		Btn_Step_Diag				:sButtonVisu_Tree;
		Btn_Lng					:sButtonVisu_Tree;

		Btn_VisuBeenden			:sButtonVisu_Tree;
END_STRUCT
END_TYPE

(* Data type in System/Error_and_Message *)
TYPE sMessageLine :
STRUCT
	Visible				: BOOL;
	Editable			: BOOL;
	Text		    	: STRING(80);
	MsgTypeEnum		: eMsgDataLineType; (*BOOL, DINT, REAL, STRING *)
	MsgType				: STRING; (*BOOL, DINT, REAL, STRING *)
	MsgBool	  	  : BOOL;
	MsgInt		    : DINT;
	MsgReal			  : REAL;
	MsgString			: STRING(40);
END_STRUCT
END_TYPE

(* Data type in System/Error_and_Message *)
TYPE sMessageText :
STRUCT
	ShowMessage				: BOOL;
	ID							: STRING(20);
	Name						: STRING(30);
	Text						: STRING(160);
	Color						: DINT; (*from STRUCT Colors*)
	DateTime					: DT;
	Station						: DINT;
	Button1						: sButtonVisu;
	Button2						: sButtonVisu;
END_STRUCT
END_TYPE

(* Data type in System/Error_and_Message *)
TYPE sMessageVisu :
STRUCT
	ShowMessage			: BOOL;
	ID						: STRING(20);
	Name					: STRING(30);
	Text					: STRING(255);
	Color					: DINT; (*from STRUCT Colors*)
	DateTime				: DT;
	Station					: DINT;
	Button1					: sButtonVisu;
	Button2					: sButtonVisu;
	MessageLine			: ARRAY [1..10] OF sMessageLine;

	BtnHide					: sButtonVisu;
	BtnShow					: sButtonVisu;
	TextMinimized			: STRING(60);
END_STRUCT
END_TYPE

(* Data type in System/VisuInterface *)
TYPE sModeSelectInit :
STRUCT
	(* Structure for initialising the object *)
	(* Initialisierungsstruktur des Objektes *)

	InstName							:	STRING(16);		(* Instanzname of the object *)
																				(* Name der Instanz *)
	EnableQuickAutoStart 	: BOOL;     		(* If TRUE, then show AutoStartButton in MODE_AUTO always:
                                    			          if HomePosition=FALSE then change first in MODE=MODE_HOME_POS_RUN *) 
	RemoteAutoStopToManual: BOOL;     		(* If TRUE, then the mode change to MODE=MODE_MANUAL
                                   				          if FALSE then change to MODE=MODE_AUTO_STOP *) 

	HideManualButton			:	BOOL;     		(* If TRUE, then hide ManualMode-Button (then ManuelMode is not used)*)
	HideNextStepButton		:	BOOL;     		(* If TRUE, then hide StepMode-Button (then StepMode is not used)*)
END_STRUCT
END_TYPE

(* Data type in System/VisuInterface *)
TYPE sModeSelectVisu :
STRUCT

	BtnManual		: sButtonVisu;
	BtnStep			: sButtonVisu;
	BtnStepCycle: sButtonVisu;
	BtnAuto			: sButtonVisu;
	BtnAutoStart: sButtonVisu;
	BtnAutoStop	: sButtonVisu;
	BtnRunEmpty	: sButtonVisu;
	BtnHomeRun	: sButtonVisu;
	BtnSpecial	: sButtonVisu;
	BtnSpecStep	: sButtonVisu;
	BtnReset		: sButtonVisu;

	ManualOn					:	BOOL;		(*manual-mode is activ*)
	StepOn						:	BOOL;		(*step-mode is activ*)
	AutoOn						:	BOOL;		(*auto-mode is activ*)
	AutoStartOn				:	BOOL;		(*automatic is running*)
	AutoStopOn				:	BOOL;		(*automaticv running in last cycle*)
	RunEmptyOn				:	BOOL;		(*machine is running empty*)
	HomePosRunOn			:	BOOL;		(*home-position-run is activ*)
	SpecialOn					:	BOOL;		(*special-mode is activ*)

	BasicManualMode		:	BOOL;		(*the basic-mode 'manual' is activ*)
	BasicAutoMode			:	BOOL; 	(*the basic-mode 'automatic' is activ*)
															(*auto, autostart, autostop, step, homeposrun*)
	HomePositionOk		:	BOOL;		(* home position *)
	HomePositionInfoNo: DINT;		(* missing to home position *)
	DisableString			: STRING(50);	(* string shows missing signal *)
															(* string zeigt fehlende Bedingung an *)
	State							:	DINT;		(*status-messages from mode-dispatcher*)
END_STRUCT
END_TYPE

(* Data type in System/MP_ShiftHandler *)
TYPE sMP_ShiftData :
STRUCT
	ShiftName			: STRING;
	ShiftIndex		: DINT;
	ShiftActive		: BOOL;
	TimeStart			: Timestruct;
	TimeEnd				: Timestruct;

END_STRUCT
END_TYPE

(* Data type in System/MP_ShiftHandler *)
TYPE sMP_ShiftHandler :
STRUCT
	ActiveShift	:	sMP_ShiftData;
	Shift				: ARRAY[1..3] OF sMP_ShiftData;
END_STRUCT
END_TYPE

(* Data type in System/MachineParameterHandler *)
TYPE sMPHandler :
STRUCT

	FileListExport				: ARRAY[1..20] OF STRING(80);
	FileListLocal					: ARRAY[1..20] OF STRING(80);

	FileNameSelected			: STRING(80);
	FileNameSaveAs			: STRING(80);

	FileIndex					: DINT;
	FileFilter						: STRING(80);

	FileListUpdate				: BOOL;

	BtnImport					: sButtonVisu;
	BtnExport					: sButtonVisu;

	MessageString				: STRING;

END_STRUCT
END_TYPE

(* Data type in System/LoginDialog *)
TYPE sNumericKeypad :
STRUCT
		Visible					:	BOOL;
		Enable					:	BOOL;

		btn_Key1						:	sButtonVisu;
		btn_Key2						:	sButtonVisu;
		btn_Key3						:	sButtonVisu;
		btn_Key4						:	sButtonVisu;
		btn_Key5						:	sButtonVisu;
		btn_Key6						:	sButtonVisu;
		btn_Key7						:	sButtonVisu;
		btn_Key8						:	sButtonVisu;
		btn_Key9						:	sButtonVisu;
		btn_Key0						:	sButtonVisu;
		btn_KeyDot					:	sButtonVisu;

		btn_KeyBack					:	sButtonVisu;
		btn_KeyEsc					:	sButtonVisu;
		btn_KeyClear				:	sButtonVisu;
		btn_KeyOK 					:	sButtonVisu;
		btn_KeyVorzeichen		:	sButtonVisu;


		InputString			:	STRING;

END_STRUCT
END_TYPE

(* Data type in sStation/sPersistent *)
TYPE sPersDaten :
STRUCT

	i_DayOfYearAutoCheckIn	:DINT;

END_STRUCT
END_TYPE

(* Data type in sStation/sTurnTable *)
TYPE sProcessData :
STRUCT

	Nest_Nr			: DINT;
	Part				: BOOL;
	Result 			: DINT;					(*   0 = Teil noch nicht bearbeitet bzw. Nest leer*)
											(*   1 =  Oberseite OK*)
											(*  11 = Oberseite und Unterseite OK*)
											(*  99 = Teil ist NOK	*)
END_STRUCT
END_TYPE

(* Data type in zLibrary/EsponRobot/Drives_IO *)
TYPE sSMCGlobalVar :
STRUCT
 ObjCount			: INT 					:=0;
END_STRUCT
END_TYPE

(* Data type in zLibrary/EsponRobot/Drives_IO *)
TYPE sSMCInit :
STRUCT
	InstName					:	STRING(20);	(* Instance name of the object *)
	Description				:	STRING(50);	(* Description of instance     *)
	MaxTime						:	DINT; 			(* number of 100ms cycles to Timeout *)
	StepDataFilePath	:	STRING(80);	(* path for pos. file from ACT Controller export *)
END_STRUCT
END_TYPE

(* Data type in zLibrary/EsponRobot/Drives_IO *)
TYPE sSMCPosStruct :
STRUCT
	MoveFct 					:	STRING(8);
	PosValue  				:	REAL;
END_STRUCT
END_TYPE

(* Data type in zLibrary/EsponRobot/Drives_IO *)
TYPE sSMCVisu :
STRUCT
(* EA's from Axis *)
	In_Busy           : BOOL;
	In_Area           : BOOL;
	In_SetupOk        : BOOL;
	In_InPosition     : BOOL;
	In_Ready          : BOOL;
	In_EstopOk        : BOOL;
	In_NoAlarm        : BOOL;
	qRelease          : BOOL;
	qStepDataNo_0     : BOOL;
	qStepDataNo_1     : BOOL;
	qStepDataNo_2     : BOOL;
	qStepDataNo_3     : BOOL;
	qStepDataNo_4     : BOOL;
	qStepDataNo_5     : BOOL;
	qSetup            : BOOL;
	qMoveHold         : BOOL;
	qMoveStart        : BOOL;
	qReset            : BOOL;
	qServoOn          : BOOL;

(* Outputvariables*)
	State								: DINT;					(* State of the valve												*)
	HomePosition				: BOOL; 				(* valve in home-position										*)
	ErrorString					: STRING(40);		(* string shows missing signal 							*)
	InstName						:	STRING(20);		(* Instance name of the object *)
	Description					:	STRING(40);		(* Description of instance     *)
	ProcessTime					: DINT;					(* Process time *)
	PosArray						: ARRAY [0..63] OF sSMCPosStruct;
	ShowPosArray				: BOOL;

(* From Visu to Object *)
	PosNo								:	DINT;					(* Position No from Robot *)

	BtnRelease					:	sButtonVisu;	(* Manage button *)
	BtnSetup						:	sButtonVisu;	(* Manage button *)
	BtnMoveHold					:	sButtonVisu;	(* Manage button *)
	BtnMoveStart				:	sButtonVisu;	(* Manage button *)
	BtnReset    				:	sButtonVisu;	(* Manage button *)
	BtnServoOn  				:	sButtonVisu;	(* Manage button *)
	BtnReadFile  				:	sButtonVisu;	(* Manage button *)
END_STRUCT
END_TYPE

(* Data type in sStation/sTurnTable *)
TYPE sStationData :
STRUCT
	Description				: STRING:='';
	HomePos				: BOOL;
	Activated				: BOOL := TRUE; (* Station Deactivated *)
	CycleTime				: DINT;

	ProcessData			: sProcessData; (*is shifted when Table turns*)
END_STRUCT
END_TYPE

(* Data type in EPT Lib/Achsen/EL72x1 *)
TYPE st_config_axis :
STRUCT
	Description				:STRING;
	InstName				:STRING;
	Aktiv					:BOOL;
	Skalierfaktor				:LREAL;
	Bit_Geber				:INT;
	Getriebefaktor			:LREAL;
	Modulo					:BOOL:=TRUE;
	Pos_Faktor				:LREAL;						(*Weg bei einer Motorumdrehung in mm*)
	ModeOfOperation			:enum_ModeOfOperation:=CSP;
	maxRpm					:INT;				(*Maximale Drehzahl des Motor*)
(*nur für Coe-Online 7010.03 (CSP) position mode*)

	RampTime				:TIME;				(*Baustelle*)(*Beschleunigungszeit und Bremsrampe*)
	PosDiffControl_on			:BOOL;				(*Baustelle*)
	max_PosDiff				:LREAL;				(*Baustelle*)
	UeberlaufControl_on		:BOOL;
	Torque_Limit				:INT;				(*bei 0 ausgeschaltet*)(* Baustelle*)
	SW_Limit_on				:BOOL;
	SW_Limit_min			:LREAL;
	SW_Limit_max			:LREAL;
	lr_kp 					:LREAL := 800;
	lr_ki 						:LREAL := 100.0;
	lr_kd 					:LREAL := 50;
END_STRUCT
END_TYPE

(* Data type in zLibrary/KeyenceEtherCat *)
TYPE st_config_Keyence :
STRUCT
	Description				:STRING;
	InstName				:STRING;
	Aktiv					:BOOL;
END_STRUCT
END_TYPE

(* Data type in EPT Lib/Achsen/EL72x1 *)
TYPE st_ctrl_Axis :
STRUCT
	in		: st_ctrl_in_axis;
	out		: st_ctrl_out_axis;
END_STRUCT
END_TYPE

(* Data type in EPT Lib/Achsen/EL72x1 *)
TYPE st_ctrl_in_axis :
STRUCT
	Position					:LREAL;

(*Bit 0*) Ready_to_switch_on	:BOOL;
(*Bit 1*) Switched_on			:BOOL;
(*Bit 2*) Operation_enabled		:BOOL;
(*Bit 3*) Fault					:BOOL;
(*Bit 4 : reserved*)
(*Bit 5 : reserved*)
(*Bit 6*) Switch_on_disabled		:BOOL;
(*Bit 7*) Warning				:BOOL;
(*Bit 8 + 9 : reserved*)
(*Bit 10*) TxPDOToggle		:BOOL; (*An-/Abwahl über 0x8010:01[} 136]*)
(*Bit 11*) Internal_Limit_active	:BOOL;
(*Bit 12*) Target_value_ignored	:BOOL;
(*Bit 13 - 15 : reserved*)

	Velocity				:LREAL;
	Following_Error		:LREAL;

END_STRUCT
END_TYPE

(* Data type in EPT Lib/Achsen/EL72x1 *)
TYPE st_ctrl_out_axis :
STRUCT
	Target_Position		:LREAL;
	Tearget_Velocity		:DINT;

(*Bit 0*)	Switch_on					:BOOL;
(*Bit 1*)	Enable_voltage		:BOOL;
(*Bit 2	*)Shutdown					:BOOL;
(*Bit 3*)	Enable_operation	:BOOL;
(*Bit 4 - 6 : reserved*)
(*Bit 7*)	Fault_reset				:BOOL;
(*Bit 8 - 15 : reserved*)

END_STRUCT
END_TYPE

(* Data type in zLibrary/KeyenceEtherCat *)
TYPE st_ctrl_out_Keyence :
STRUCT
			iJobNo					:INT;

(*Bit 0*)	bReset					:BOOL;	(*Reserviert (alles zurücksetzen)*)
(*Bit 1*)	bPrgChange				:BOOL;	(*Programmwechselanforderung*)
(*Bit 2*)	bTrigger				:BOOL;	(*Trigger*)

(*nicht benutzt*)
(*Bit 3*) 	bMaster					:BOOL;	(*Master-Registrierunganforderung *)
(*Bit 4*) 	bSpeicherstopp			:BOOL;	(*Speicherstopp SD-Karte Anfrage*)
(*Bit 5*) 	bStatistikruecksetzung	:BOOL;	(* Statistikrücksetzung anfordern*)
(*Bit 6*) 	bFehlerLoeschen			:BOOL;	(*Anforderung Fehler löschen*)
(*Bit 7*) 	OCR_Seriennummer		:BOOL;	(*Anforderung OCR-Seriennummer Hochzählen*)
(*Bit 8*) 	Zaehlung_Ruecksetzen	:BOOL;	(*Zählung-Rücksetzen Anforderung*)
(*Bit 9*) 	Statistik_Ruecksetzen	:BOOL;	(*Anforderung Statistik aller Programme Rücksetzen*)
(*Bit 10*) 	Reserviert_10			:BOOL;	(**)
(*Bit 11*) 	Reserviert_11			:BOOL;	(**)
(*Bit 12*) 	Reserviert_12			:BOOL;	(**)
(*Bit 13*) 	Reserviert_13			:BOOL;	(**)
(*Bit 14*) 	Reserviert_14			:BOOL;	(**)
(*Bit 15*) 	Reserviert_15			:BOOL;	(**)


(*
DL-EC1A: PDO-Kommunikation (Prozessdaten-Objekte)

	Daten Senden via anInputRequest (* Index: 16#7000; SubIndex: 16#0001 - 16#0005 *)

	Index: 16#7000  SubIndex: 16#0001
		Inhalt:
			Bit 0 = Reserviert (alles zurücksetzen)
			Bit 1 = Programmwechselanforderung
			Bit 2 = Trigger
			Bit 3 = Master-Registrierunganforderung 
			Bit 4 = Speicherstopp SD-Karte Anfrage 
			Bit 5 = Statistikrücksetzung anfordern 
			Bit 6 = Anforderung Fehler löschen 
			Bit 7 = Anforderung OCR-Seriennummer Hochzählen 
			Bit 8 = Zählung-Rücksetzen Anforderung 
			Bit 9 = Anforderung Statistik aller Programme Rücksetzen
			Bit 10-15 = Reserviert
	Index: 16#7000  SubIndex: 16#0002
		Inhalt:
			Bit 0 = Reserviert	 (alles zurücksetzen)
			Bit 1 = Programmnummer ändern (Bit 0)
	Index: 16#7000  SubIndex: 16#0003
		Inhalt:
			Bit 0 = Reserviert  (alles zurücksetzen)
			Bit 1 = Programmnummer ändern (Bit 1)
	Index: 16#7000  SubIndex: 16#0004
		Inhalt:
			Bit 0 = Reserviert  (alles zurücksetzen)
			Bit 1 = Programmnummer ändern (Bit 2)
	Index: 16#7000  SubIndex: 16#0005
		Inhalt:
			Bit 0 = Reserviert
			Bit 1 = Programmnummer ändern (Bit 3)
*)

END_STRUCT
END_TYPE

(* Data type in EPT Lib/Achsen/EL72x1 *)
TYPE st_fb_axis :
STRUCT
	ton_uez			:TON;
	ton_uez_velo	:TON;
	ton_quitt		:TON;
	ton_aufPos		:TON;
	ton_Busy		:TON;


	r_trig_stop		: R_TRIG;
	r_trig_quitt	: R_TRIG;
	r_trig_reset	: R_TRIG;
	r_trig_jogP		: R_TRIG;
	r_trig_jogM		: R_TRIG;
	r_trig_MoveP	: R_TRIG;
	r_trig_MoveM	: R_TRIG;
	r_trig_MotorOn	: R_TRIG;
	r_trig_MoveAbs	: R_TRIG;

	r_trig_teach		: R_TRIG;
	r_trig_kont			: R_TRIG;
	r_trig_ink_10		: R_TRIG;
	r_trig_ink_100		: R_TRIG;
	r_trig_ink_1000		: R_TRIG;
	r_trig_ink_var		: R_TRIG;
	r_trig_Auto			: R_TRIG;
	r_trig_Hand			: R_TRIG;
END_STRUCT
END_TYPE

(* Data type in EPT Lib/Achsen/EL72x1 *)
TYPE st_Help_axis :
STRUCT
	b_init				:BOOL;
	b_init2				:BOOL;
	b_ToggleHelp		:BOOL;

	b_Pos_nr_Empty		:ARRAY [-1..NO_OF_POS_AXIS] OF BOOL;
	PosNr				:INT:=1;
	Pos					:LREAL;

END_STRUCT
END_TYPE

(* Data type in EPT Lib/Achsen/EL72x1 *)
TYPE st_PID_axis :
STRUCT
	lr_Override			:LREAL;

	lr_delta				: LREAL := 0.0;
	lr_delta_alt			: LREAL := 0.0;
	lr_delta_dif			: LREAL := 0.0;

	lr_current_p			: LREAL := 0.0;
	lr_current_i			: LREAL := 0.0;
	lr_current_d			: LREAL := 0.0;

	lr_current_v			: LREAL := 0.0;
	lr_tmp				: LREAL := 0.0;

	lr_delta_targetpos	: LREAL := 0.0;
	lr_targetpos_alt		: LREAL := 0.0;

END_STRUCT
END_TYPE

(* Data type in EPT Lib/Achsen/EL72x1 *)
TYPE st_Pos :
STRUCT
	Description		: STRING;
	Pos	 			: LREAL;
END_STRUCT
END_TYPE

(* Data type in EPT Lib/Achsen/EL72x1 *)
TYPE st_Pos_axis :
STRUCT
	ist					:REAL;
	soll					:REAL;
	r_18bit				:REAL;
	r_20bit				:REAL;
	r_32bit				:REAL;

	lr_DiffPuls			:LREAL := 0.0;
	lr_DiffVelo			:LREAL := 0.0;
	lr_MaxDiff			:LREAL := 0.0;

	(*Überlauf*)
	lr_akt_alt				:LREAL;
	lr_delta_ueberlauf		:LREAL;
	i32_count_ueberlauf	:DINT;
	lr_Uebrlauf_DistOne	:LREAL;
	lr_Uebrlauf_Dist		:LREAL;

	(*Singelturn*)
	lr_ModuloPosInc		:LREAL;
	lr_ModuloHelp		:LREAL;
	lr_ModuloHelp2		:LREAL;
	i16_ModuloHelp		:INT;
	lr_ModuloCount		:LREAL;

	(*Multiturn*)
	lr_Pos				:LREAL;
	lr_Target				:LREAL;
	lr_Mod				:LREAL;

	lr_Offset_Ink			:LREAL;
	i32_Offset_Ink			:UDINT;

END_STRUCT
END_TYPE

(* Data type in EPT Lib/Achsen/EL72x1 *)
TYPE st_sdo :
STRUCT
	fb_ec_coe_sdo_write_ex		: FB_EcCoESdoWriteEx;
	fb_ec_coe_sdo_read_ex		: FB_EcCoESdoReadEx;

(*	st_eccoe_sdo				:struct_eccoe_sdo;*)

	s_SlaveNetId 			: T_AmsNetId := '';
	ui16_SlaveAddr 			: UINT := 0;			 (* Address of the slave device.*)
	i8_SubIndex 			: BYTE := 0;			 (* CANopen Sdo subindex.*)
	w_Index 				: WORD := 16#00;	 (* CANopen Sdo index.*)

	acObjectData				:ARRAY[0..MAX_STRING_LENGTH] OF BYTE;

END_STRUCT
END_TYPE

(* Data type in EPT Lib/Achsen/EL72x1 *)
TYPE st_sm_axis :
STRUCT
	sm_timeout			:BOOL;
	sm_Error_Klemme	:BOOL;
	sm_Error_Warnung	:BOOL;
	sm_PosDiff			:BOOL;
	sm_Check_Velo		:BOOL;
	sm_SW_Limit			:BOOL;
	sm_fehler_daten_schreiben:BOOL;
	sm_connect			:BOOL;
	sm_Ueberlauf		:BOOL;
	sm_Torque_zu_gross	:BOOL;
	sm_NotausNok		:BOOL;
	sm_Move				:BOOL;
END_STRUCT
END_TYPE

(* Data type in EPT Lib/Achsen/EL72x1 *)
TYPE st_Velo_axis :
STRUCT
	maxRpmNachGertiebe	:LREAL;	(*Maximale Drehzahl nach Getriebe*)
	maxLinear		:LREAL;	(*Maximale Geschwindigkeit in mm/min*)
	maxRpm				:LREAL;	(*in U/min oder in mm/min*)
	Vorgabe_Velo_rpm	:LREAL;	(*in U/min*)
	sollRpm				:LREAL;	(*in U/min*)
	soll					:LREAL;
	ist				:LREAL;
	dif				:LREAL;
	Faktor			:LREAL;

END_STRUCT
END_TYPE

(* Data type in EPT Lib/Achsen/EL72x1 *)
TYPE st_Visu_axis :
STRUCT
	Einheit_pos			:STRING(10);
	Einheit_velo			:STRING(10);

	BtnReset			: sButtonVisu;
	BtnStop				: sButtonVisu;
	BtnJogP			: sButtonVisu;
	BtnJogM			: sButtonVisu;
	BtnMotorOn			: sButtonVisu;
	BtnMoveAbs		: sButtonVisu;
	BtnTeach			: sButtonVisu;

	PosNr				:INT:=1;
	Poslist				:BOOL;

	Control				:BOOL;
	b_kont				:BOOL;
	b_ink_10			:BOOL;		(*in µm*)
	b_ink_100			:BOOL;		(*in µm*)
	b_ink_1000			:BOOL;		(*in µm*)
	b_ink_var			:BOOL;		(*in mm variabel *)
	lr_ink_var			:LREAL:=10;

	b_Pos_nr			:ARRAY [-1..NO_OF_POS_AXIS] OF BOOL;
	b_PosNr			:BOOL;
END_STRUCT
END_TYPE

(* Data type in System/GlobalStates *)
TYPE StateMode :
(
(* different modes of the Mode-Dispatcher
   verschiedene Betriebsarten des Betriebsartenbausteines *)
	MODE_NON					:= 0,		(*MODE_NON*)
	MODE_MANUAL				:= 10,		(*MODE_MANUAL*)
	MODE_STEP					:= 20,		(*MODE_STEP*)
	MODE_STEP_RUN				:= 21,		(*MODE_STEP_RUN*)
	MODE_STEP_STOP			:= 22,		(*MODE_STEP_STOP*)
	MODE_AUTO					:= 30,		(*MODE_AUTO*)
	MODE_AUTO_RUN				:= 31,		(*MODE_AUTO_RUN*)
	MODE_AUTO_STOP 			:= 32,		(*MODE_AUTO_STOP*)
	MODE_HOME_POS_RUN		:= 40,		(*MODE_HOME_POS_RUN*)
	MODE_SPECIAL				:= 50 		(*MODE_SPECIAL*)
);
END_TYPE

(* Data type in System/GlobalStates *)
TYPE StateObject :
	(
	STATE_ERROR			:= -1,  		 (*STATE_ERROR Objekt meldet Fehler *)
	STATE_TIMEOUT  		:= -2,	 	  (*STATE_TIMEOUT Objekt meldet Fehler *)
	STATE_UNDEFINED		:= 0,		(*STATE_UNDEFINED Das Objekt befindet sich in einem undefinierten Zustand *)
	STATE_OK			:= 1,		(*STATE_OK Die letzte Aktion wurde erfolgreich durchgeführt *)
	STATE_RUN			:= 2,		(*STATE_RUN Die Aktion wird gerade durchgeführt *)
	STATE_WAIT			:= 3,		(*STATE_WAIT Bereit (für neue Aktion) *)
	STATE_STOPPED		:= 4,		(*STATE_STOPPED Objekt gesperrt(durch externes Enable) *)
	STATE_RESETS		:= 5,		(*STATE_RESETS Objekt wird zurückgesetzt *)
	STATE_IGNORED		:= 6 		(*STATE_IGNORED Alle Stati und Meldungen werden ignoriert *)
	);
END_TYPE

(* Data type in System/GlobalStates *)
TYPE StateResult :
(
	RESULT_NON 			:=	0,  (* No Result from sequence *)
	RESULT_OK			:=	1,	(* End of Sequence with OK *)
	RESULT_NOK			:=	2,	(* End of Sequence with NOT OK *)
	RESULT_REW			:=	3 	(* End of Sequence with REWORK *)

);
END_TYPE

(* Data type in System/TypeDataHandler *)
TYPE sTDHandler :
STRUCT
	TypeDataValid			: BOOL;

	FileList					: ARRAY[1..NO_OF_FILES] OF STRING(80);
	FileNameSelected		: STRING(80);
	FileNameSaveAs		: STRING(80);

	FileListUpdate			: BOOL;
	FileIndex				: DINT:=1;
	FileFilter					: STRING(80);

	BtnLoad				: sButtonVisu;
	BtnSave				: sButtonVisu;
	BtnSaveAs				: sButtonVisu;
	BtnActivate				: sButtonVisu;
	BtnClose				: sButtonVisu;
	BtnDelete				: sButtonVisu;
	BtnNew					: SButtonVisu;

END_STRUCT
END_TYPE

(* Data type in EPT Lib/Allgemeine Kontrollstrukturen Objekte *)
TYPE struct_config :
STRUCT
	str_instanz_name					: STRING(48) := '';
	str_beschreibung					: STRING(50) := '';
	b_station_aktiv					: BOOL := FALSE;
	b_station_in_simulation				: BOOL := FALSE;
	i16_meld_startindex				: INT := 0;
	b_config_fertig					: BOOL := FALSE;
END_STRUCT
END_TYPE

(* Data type in EPT Lib/Allgemeine Kontrollstrukturen Objekte *)
TYPE struct_ctrl :
STRUCT
	in		: struct_ctrl_in;
	out		: struct_ctrl_out;
END_STRUCT
END_TYPE

(* Data type in EPT Lib/Allgemeine Kontrollstrukturen Objekte *)
TYPE struct_ctrl_in :
STRUCT
	b_quitt						: BOOL := FALSE;
	b_stop 						: BOOL := FALSE;
         b_halt		  	 			: BOOL := FALSE;
         b_definierter_halt  	 			: BOOL := FALSE;
	b_init 						: BOOL := FALSE;
	b_init_2 						: BOOL := FALSE;
         b_preinit                				: BOOL := FALSE;
	b_start						: BOOL := FALSE;
	b_start_2						: BOOL := FALSE;
	b_gutteil_produziert 			: BOOL := FALSE;
	b_schlechtteil_produziert 		: BOOL := FALSE;
	b_start_lesen					: BOOL := FALSE;
	b_start_schreiben				: BOOL := FALSE;
	b_schutzhaube_ab			: BOOL := FALSE;
	b_schutzhaube_auf			: BOOL := FALSE;
	b_nachtabschaltung			: BOOL := FALSE;
	b_gehe_step_ibn				: BOOL := FALSE;
	b_ibn_start					: BOOL := FALSE;
	b_freigabe					: BOOL := FALSE;
END_STRUCT
END_TYPE

(* Data type in EPT Lib/Allgemeine Kontrollstrukturen Objekte *)
TYPE struct_ctrl_out :
STRUCT
	b_bereit 						: BOOL := FALSE;
	b_bereit_2					: BOOL := FALSE;
         b_prebereit               			: BOOL := FALSE;
	b_fehler 						: BOOL := FALSE;
	b_fertig						: BOOL := FALSE;
	b_fertig_2					: BOOL := FALSE;
	b_bandende					: BOOL := FALSE;
	b_kontroller_start				: BOOL := FALSE;
	b_gestoppt					: BOOL := FALSE;
	b_angehalten					: BOOL := FALSE;
	b_haube_oeffnen				: BOOL := FALSE;
	b_nachtabschaltung			: BOOL := FALSE;
	b_einzelfertigung				: BOOL := FALSE;
	b_busy						: BOOL := FALSE;
 st_takt_Time : STRING;
END_STRUCT
END_TYPE

(* Data type in sStation/sMachineParameter/Service *)
TYPE struct_daten_service :
STRUCT
	Name			: STRING(255);
	Default_Value	: LREAL;
	Current_Value	: LREAL;
	Warning_Value	: LREAL;
	Warning_reached	: BOOL:= FALSE;
	Default_reached	: BOOL:= FALSE;
	Type_Service	: eService_Type;
	Unit				: STRING(20);
	Starttag			: INT := 0;
	Startstunden	: LREAL := 0;
	StartBetriebsStd	: LREAL := 0;
END_STRUCT
END_TYPE

(* Data type in EPT Lib/Achsen/BECKHOFF *)
TYPE struct_eccoe_sdo :
STRUCT
	s_ec_slave_net_id 		: T_AmsNetId := '';
	ui16_slave_addr 			: UINT := 0; (* Address of the slave device.*)
	i8_sub_index 				: BYTE := 0; (* CANopen Sdo subindex.*)
	w_index 					: WORD := 16#00; (* CANopen Sdo index.*)
	dw_p_source_buffer 		: DWORD := 16#0000; (* Contains the address of the buffer containing the data to be send. *)
	dw_p_destination_buffer	: DWORD := 16#0000; (* Contains the address of the buffer for the received data. *)
	ui32_buffer_length 			: UDINT := 0; (* Contains the max. number of bytes to be received. *)
	ui32_value 				: UDINT := 0; (* variable to be written to the CoE Object *)
	ui16_value 				: UINT := 0; (* variable to be written to the CoE Object *)
	byte_value 				: BYTE := 16#00; (* variable to be written to the CoE Object *)
	bool_value 				: BOOL := FALSE; (* variable to be written to the CoE Object *)
END_STRUCT
END_TYPE

(* Data type in EPT Lib/Hydra *)
TYPE struct_Hydra :
STRUCT
	s_Start_Time	: STRING(20) := '01.01.1970 00:00:00';	(* TT.MM.JJJJ HH:MM:SS *)
	i_Counter		: ARRAY[1..104] OF DINT;	(* alle Zähler 4-stellig *)
	b_Input		: ARRAY[1..128] OF BOOL:=128(FALSE);
END_STRUCT
END_TYPE

(* Data type in EPT Lib/Hydra *)
TYPE struct_Hydra8 :
STRUCT
	iCounter		: ARRAY[1..20] OF DINT;	(* alle Zähler 4-stellig *)
	bStatus		: ARRAY[1..999] OF BOOL:=999(FALSE);	(* TRUE wenn Status aktiv ist *)
END_STRUCT
END_TYPE

(* Data type in EPT Lib/Allgemeine Kontrollstrukturen Objekte *)
TYPE struct_objekt :
STRUCT
	st_config		: struct_config;
	st_ctrl		: struct_ctrl;
END_STRUCT
END_TYPE

(* Data type in sStation/sMachineParameter/Service *)
TYPE struct_visu_service :
STRUCT
	BtnReset			: sButtonVisu;
	BtnStart			: sButtonVisu;
	BtnType			: sButtonVisu;
	Current_Value	 : STRING(20);
	Current_Value_Color	: DINT;

END_STRUCT
END_TYPE

(* Data type in sStation/sTypedata *)
TYPE sTypeData :
STRUCT
	(* allegmeine Typinfos *)
	ArtNo					: STRING(30); (* interne Kundenartikelnummer *)
	TypeName				: STRING(30); (* xml-Dateiname *)
	TypeDescription			: STRING(30); (* Typbeschreibung optional *)

	(* Typmerkmale *)
	TypeCode				: STRING(5); (* Typkennung z.B. P310 *)

	Override_Band			: INT:=20; (* *)
	Override_Robi			: INT:=20; (* *)

	PosAbstapeln	 		: ARRAY [1..NO_OF_POS_AXIS] OF st_Pos;	(*	1=unten, 2= mitte, 3=oben*)
	PosAufstapeln	 		: ARRAY [1..NO_OF_POS_AXIS] OF st_Pos;	(*	1=unten, 2= mitte, 3=oben*)
	PosTrayAusheben	 		: ARRAY [1..NO_OF_POS_AXIS] OF st_Pos;	(*	1=unten, 2=oben*)

	TestpartBilister		: BOOL;
	DistIso					: LREAL;

	IFM_Positon_Dummy 		: LREAL ;
	SensopartErgebnis			: STRING(15); (*Ergebnis Sensopart Kamera*)
	Sensopart2Ergebnis			: STRING(15); (*Ergebnis Sensopart Kamera*)
	NoOfPalletsPerStack		: DINT:=1;

	(*Aus Load Info*)
	RobotOffset				: DINT;

	PartsInBlisterInlet		: DINT; (* Anzahl Teile pro Blister Einlauf *)
	PartsInRoboGripper		: DINT:=1; (* Anzahl Teile pro Robi Greifer *)

	IFM_CamProgNo			: BYTE;
	Sensopart_CamProgNo		: BYTE;
	Sensopart2_CamProgNo		: BYTE;
	Keyence_CamProgNo		: BYTE;

END_STRUCT
END_TYPE

(* Data type in System/LoginDialog *)
TYPE sUserData :
STRUCT
	UserName						: STRING;
	UserPassword					: STRING;
	UserLevel						: INT;
	UserCanChangeOwnPassword		: BOOL;
END_STRUCT
END_TYPE

(* Data type in sStation/sUserList *)
TYPE sUserList :
STRUCT
  	UserList							:	ARRAY [1..NO_OF_USERS] OF sUserData;
END_STRUCT
END_TYPE

(* Data type in zLibrary/Valve *)
TYPE sValveGlobalVar :
STRUCT
 ObjCount			: INT 					:=0;
END_STRUCT
END_TYPE

(* Data type in zLibrary/Valve *)
TYPE sValveHome :
(
	HOME_INIT		:=0,
	HOME_WORK 	:=1,
	HOME_BOTH   :=2,
	HOME_ALWAYS :=3
);
END_TYPE

(* Data type in zLibrary/Valve *)
TYPE sValveInit :
STRUCT
(* Structure for initialising a valve *)
	BitName				: STRING(25);	(* Name of bit *)
	InstName				: STRING(25);	(* Instance name of the object *)
	Description				: STRING(50);	(* Description of instance     *)
	WorkDescription			: STRING;		(* Description of work movement for e.g. down	*)
	InitDescription			: STRING;		(* Description of init movement for e.g. up   *)

	KindOfValve				: STRING;		(* kind of the valve:				A, B, D, G*)
	HomePosDefine			: DINT;			(* home-position is definded in:			 				*)
																(* 0: InitPosition, 1: WorkPosition, 2: Both  *)
	MaxTime				: DINT; 			(* number of 100ms cycles to Timeout 				  *)
	DampBothTime			: DINT; 			(* time in msec. for damp both msec  					*)
	DisableSignalMonitoring 	: BOOL; 		(* Disable signalmonitoring after movement*)
END_STRUCT
END_TYPE

(* Data type in zLibrary/Valve *)
 TYPE sValveSensor_SensorOut :
STRUCT
	SensorName				:	STRING;	(* From Sensor: Sensorname *)
	SensorSignal			:	BOOL;		(* From Sensor *)
	SensorType				: sValveSensorType; (* From Sensor: Init- Or Worksensor *)
END_STRUCT
END_TYPE

(* Data type in zLibrary/Valve *)
 TYPE sValveSensor_ValveOut :
STRUCT
	SignalLoExpected	: BOOL; (* From Valve: If Sensor not Low Raise Error!  *)
	SignalHiExpected	: BOOL;	(* From Valve: If Sensor not High Raise Error!  *)
END_STRUCT
END_TYPE

(* Data type in zLibrary/Valve *)
TYPE sValveSensorInit :
STRUCT
(* Structure for initialising a valve *)
	BitName				: STRING(20);	(* Name of bit *)
	InstName				: STRING(20);	(* Instance name of the object *)
	Description				: STRING(50);	(* Description of instance     *)
	SensorType				: sValveSensorType;
END_STRUCT
END_TYPE

(* Data type in zLibrary/Valve *)
TYPE sValveSensorType :
(
	sValveSensorType_NotDefined		:=0,
	sValveSensorType_INIT					:=1,
	sValveSensorType_WORK 				:=2
);
END_TYPE

(* Data type in zLibrary/Valve *)
TYPE sValveVisu :
STRUCT
(* Structure for Handshake to display a valve *)
(*--------------------------------------------------------------*)
(* sInit-Datas *)
	BitName					: STRING(25);		(* Name of bit *)
	InstName				: STRING(25);		(* Instance name of the object *)
	Description				: STRING(50);		(* Description of instance     *)
	SAInitPosName			: STRING(16);		(* Name of Sensor Initpostion of cylinder A 	*)
	SAWorkPosName			: STRING(16);		(* Name of Sensor Workposition of cylinder A	*)
	SBInitPosName			: STRING(16);		(* Name of Sensor Initposition of cylinder B 	*)
	SBWorkPosName			: STRING(16);		(* Name of Sensor Workposition of cylinder B 	*)
	SCInitPosName			: STRING(16);		(* Name of Sensor Initposition of cylinder C 	*)
	SCWorkPosName			: STRING(16);		(* Name of Sensor Workposition of cylinder C 	*)
	SDInitPosName			: STRING(16);		(* Name of Sensor Initposition of cylinder D 	*)
	SDWorkPosName			: STRING(16);		(* Name of Sensor Workposition of cylinder D 	*)
	SEInitPosName			: STRING(16);		(* Name of Sensor Initposition of cylinder E 	*)
	SEWorkPosName			: STRING(16);		(* Name of Sensor Workposition of cylinder E 	*)
	WorkDescription			: STRING(16);		(* Description of work movement for e.g. down	*)
	InitDescription			: STRING(16);		(* Description of init movement for e.g. up   *)

	NoOfInitSensors			: DINT;				(* number of sensors in initposition:	0, 1 or 2, 3	*)
	NoOfWorkSensors			: DINT;				(* number of Sensors in workposition:	0, 1 or 2, 3	*)
	NoOfValveCoils			: DINT;				(* number of valvecoils:				1 or 2		*)
	KindOfValve				: STRING(4);		(* kind of the valve:				A, B, D, G, H or I  		*)
	HomePositionInfoNo 		: DINT;				(* missing to home position 									*)

(* Outputvariables*)
	State					: StateObject;		(* State of the valve*)
	HomePosition			: BOOL; 			(* valve in home-position*)
	ErrorString				: STRING(40);		(* string shows missing signal*)
	ErrorPresent			: BOOL;

(* Internal Variables*)
	AInitPosition			: BOOL; 			(* Sensor InitPosition of cylinder A*)
	AWorkPosition			: BOOL; 			(* Sensor WorkPosition of cylinder A*)
	BInitPosition			: BOOL; 			(* Sensor InitPosition of cylinder B*)
	BWorkPosition			: BOOL; 			(* Sensor WorkPosition of cylinder B*)
	CInitPosition			: BOOL; 			(* Sensor InitPosition of cylinder C*)
	CWorkPosition			: BOOL; 			(* Sensor WorkPosition of cylinder C*)
	DInitPosition			: BOOL; 			(* Sensor InitPosition of cylinder D*)
	DWorkPosition			: BOOL; 			(* Sensor WorkPosition of cylinder D*)
	EInitPosition			: BOOL; 			(* Sensor InitPosition of cylinder E*)
	EWorkPosition			: BOOL; 			(* Sensor WorkPosition of cylinder E*)
	CoilA					: BOOL; 			(* For Moving to WorkPosition*)
	CoilB					: BOOL; 			(* For Moving to InitPosition*)
	ProcessTime				: DINT;				(* Counts the time in ms*)

	BtnMoveWork				: sButtonVisu;		(* Manage button *)
	BtnMoveInit				: sButtonVisu;		(* Manage button *)
	BtnReset				: sButtonVisu;		(* Manage button *)

END_STRUCT
END_TYPE

(* Data type in sStation/sVisuInterface *)
TYPE sVisu:
STRUCT
(*---------------------------------------------------------------------------
  System
  ---------------------------------------------------------------------------*)
	ErrorHandler				: sErrorHandlerVisu;
	ErrorHistory				: sErrorHandlerVisu;
	ErrorHistoryScroll		: DINT;
	SelectPictureName		: STRING(20);
	SavePersistentData  	: BOOL;

	Message				: sMessageVisu;
	ModeSelect				: sModeSelectVisu;
	LoginHandler			: sVisuLoginDialog;
	MainMenue				: sMainMenue;

(*---------------------------------------------------------------------------
  Station00
  ---------------------------------------------------------------------------*)
	ST00_40_F1 			: sDigInVisu; (* Vorsicherungen Leistung iO *)
	ST03_210_S1 			: sDigInVisu; (* Not-Aus 1 Anlage ausgelöst *)
	ST08_210_S2 			: sDigInVisu; (* Not-Aus 2 Anlage ausgelöst *)
	ST00_X4_16	 		: sDigInVisu; (* Not-Halt 2 Tampondrucker ausgelöst *)
	ST00_200_A1_A1 		: sDigInVisu; (* Not-Aus iO *)
	ST00_220_S1	 		: sDigInVisu; (* Schutztüre 1 geöffnet *)
	ST00_220_S2	 		: sDigInVisu; (* Schutztüre 1 geöffnet *)
	ST00_230_S2_E1 		: sDigInVisu; (* Schutztüre 1 geschlossen *)
	ST00_240_S1 		: sDigInVisu; (* Schutztüre 9 geschlossen *)
	ST00_226_S1			: sDigInVisu;(*Hubtüre 1 Schleuse Einlauf STN 8 geschlossen*)
	ST00_226_S2			: sDigInVisu;(*Hubtüre 2 Schleuse Einlauf STN 8 geschlossen*)
	ST00_227_S1			: sDigInVisu;(*Hubtüre 3 Schleuse Auslauf STN 8 geschlossen*)
	ST00_227_S2			: sDigInVisu;(*Hubtüre 4 Schleuse Auslauf STN 8 geschlossen*)
	ST00_229_S1			: sDigInVisu;(*Schutztüre Einlauf Tray STN 8 geschlossen*)
	ST00_230_S1			: sDigInVisu;(*Schutztüre Auslauf Tray STN 8 geschlossen*)
	ST00_231_S1			: sDigInVisu;(*Schutztüre Panel / Rutsche STN 8 geschlossen*)
	ST00_232_S1			: sDigInVisu;(*Schutztüre 8 Auslauf Tray STN 8 geschlossen*)
	ST00_170_Motorschutz	: sDigInVisu;(*Motorschutz in Ordnung*)
	ST00_170_Thermokont	: sDigInVisu;(*Thermokontakt in Ordnung*)
	ST00_228_S1      		 : sDigInVisu;
	ST00_71_X1_3  		: sDigInVisu; (* Schnittstelle Bedrucken Tinte JSK auf Übergabeposition *)
	ST00_71_X1_4  		: sDigInVisu; (* Schnittstelle Bedrucken Tinte Druckstation betriebsbereit *)
	ST00_72_X1_3  		: sDigInVisu; (* Schnittstelle Tampondrucker Teil in Abholposition *)(*Band Entnahmeposition 1*)
	ST00_72_X1_8  		: sDigInVisu; (* Schnittstelle Tampondrucker Druck abgeschlossen *)
	ST00_292_S1_STOP 	: sDigInVisu; (* Bedienstelle Produktion Stop *)
	ST00_292_S2_START	: sDigInVisu; (* Bedienstelle Produktion Start *)
	ST00_292_S3_RESET	: sDigInVisu; (* Bedienstelle Produktion Reset *)
	ST00_350_B20_0 		: sDigInVisu; (* Druckschalter Wartungseinheit Hauptluft min.6 bar *)

	ST00_245_V1			: sDigOutInVisu; (* Verriegelung Schutztüren-Leuchte *)
	ST00_245_V2_START	: sDigOutInVisu; (* Bedienstelle Start-Leuchte *)
	ST00_245_V3_RESET	: sDigOutInVisu; (* Bedienstelle Reset-Schutztüren-Leuchte *)
	ST00_245_S1_STOP 	: sDigInVisu;	 (* Bedienstelle Produktion Stop *)
	ST00_245_S2_START	: sDigInVisu;	 (* Bedienstelle Produktion Start *)
	ST00_245_S3_RESET	: sDigInVisu;	 (* Bedienstelle Produktion Reset *)

	ST00_31_K1 			: sDigOutInVisu; (* Beleuchtung Anlage *)
	ST00_350_H1 			: sDigOutInVisu; (* Signalsäule RD Maschine Alarm/Störung *)
	ST00_350_H2 			: sDigOutInVisu; (* Signalsäule YE Bedienereingriff erforderlich *)
	ST00_350_H3 			: sDigOutInVisu; (* Signalsäule GN Maschine Automatik *)
	ST00_200_A1_E4 		: sDigOutInVisu; (* Quittierung Not-Aus *)
	ST00_220_S1_S31 		: sDigOutInVisu; (* Verriegelung Schutztüren *)
	ST00_292_H2_START	: sDigOutInVisu; (* Bedienstelle Start-Leuchte *)
	ST00_292_H3_RESET	: sDigOutInVisu; (* Bedienstelle Reset-Leuchte *)

	ST00_71_K2	  		: sDigOutInVisu; (* Schnittstelle Bedrucken Tinte Abholposition frei *)

	ST00_73_K2	  		: sDigOutInVisu; (* Schnittstelle allgemein Störung Tampondrucker *)
	ST00_73_K3	  		: sDigOutInVisu; (*Schnittstelle Förderband frei für Spritzmaschine*)
	ST00_73_K4	 		: sDigInVisu; 	(*Schnittstelle Freigabe von Spritzmaschine (nur für Anlagen ohne Rundtisch) *)


	ST00_74_Y2_4 : sValveVisu; (*ST00_74_Y2_4 Stopper Bandstrecke (Valve) *)
	ST00_74_Y2_5 : sValveVisu; (*ST00_74_Y2_5 Vereinzeler Bandstrecke (Valve) *)

	ST03_65_Q1			: sDigOutInVisu;		(* Kühltunnel (Lüfter)*)
	ST03_65_F1			: sDigInVisu;			(* Sicherung Kühltunnel (Lüfter)*)

(*---------------------------------------------------------------------------
  Station02
  ---------------------------------------------------------------------------*)
	ST02_FDB_55X1_5_READY 	:sDigInVisu; (* IFM Kamera Flügelerkennung links Ready *)
	ST02_FDB_55X1_6_IO			:sDigInVisu; (* IFM Kamera Flügelerkennung links Ergebnis iO *)
	ST02_FDB_55X1_6_NIO		:sDigInVisu; (* IFM Kamera Flügelerkennung links Ergebnis niO *)
	ST02_FDB_55X1_2_TRIGGER 	:sDigOutInVisu; (* IFM Kamera Flügelerkennung links Trigger *)
	ST02_FDB_55X1_7_JOB_BIT1 	:sDigOutInVisu;(* IFM Kamera links  Jobwechsel Bit 1 *)
	ST02_FDB_55X1_7_JOB_BIT2 	:sDigOutInVisu;(* IFM Kamera links  Jobwechsel Bit 2 *)

	ST02_FDB_56X1_5_READY 	:sDigInVisu; (* IFM Kamera Flügelerkennung rechts Ready *)
	ST02_FDB_56X1_6_IO			:sDigInVisu; (* IFM Kamera Flügelerkennung rechts Ergebnis iO *)
	ST02_FDB_56X1_6_NIO		:sDigInVisu; (* IFM Kamera Flügelerkennung rechts Ergebnis niO *)
	ST02_FDB_56X1_2_TRIGGER 	:sDigOutInVisu; (* IFM Kamera Flügelerkennung rechts Trigger *)
	ST02_FDB_56X1_7_JOB_BIT1 	:sDigOutInVisu;(* IFM Kamera links  Jobwechsel Bit 1 *)
	ST02_FDB_56X1_7_JOB_BIT2 	:sDigOutInVisu;(* IFM Kamera links  Jobwechsel Bit 2 *)

	ST02_S1_70K61_A1	:sDigOutInVisu; 	(* Start  Bedrucken *)

	ST02_S1_40K01 		:sDigInVisu;			(*  Freigabe Förderband von SPM *)
	ST02_FDB_80_B02 		:sDigInVisu;			(*  Band Entnahmeposition 2*)
	ST02_35_S31			:sDigInVisu; 			(* ST02 Druckschalter Wartungseinheit Hauptluft min.6 bar *)
	ST02_S1_6A01 			:sDigInVisu; 			(* ST02 Sicherung 24V *)

	ST02_FDB_40_B61	:sDigInVisu; 			(* Iso von SPM auf Band abgelegt *)
	ST02_FDB_40_B71	:sDigInVisu; 			(* Iso auf Band vor Vereinzler *)

	ST02_62_Y6			:sValveVisu; 			(*Tisch drehen 0 - 180 Grad (Valve) *)
	ST02_62_Y9			:sValveVisu; 			(*Schwenkarm 2 drehen 90 - 180 Grad (Valve) *)
	ST02_62_Y11			:sValveVisu; 			(* Schwenkarm 2 drehen 90 - 0 Grad (Valve) *)
	ST02_62_Y13			:sValveVisu; 			(*Schwenkarm 1 drehen 90 - 180 Grad (Valve) *)
	ST02_62_Y15			:sValveVisu; 			(*Schwenkarm 1 drehen 90 - 0 Grad (Valve) *)
	ST02_62_Y17			:sValveVisu; 			(*Schwenkarm 1 ISK Fixierung ein/ausfahren(Valve) *)
	ST02_62_Y18			:sValveVisu; 			(*Schwenkarm 2 ISK Fixierung ein/ausfahren(Valve) *)
	ST02_62V1				:sValveVisu; 			(* ISK Stopper ein-/ausfahren*)
	ST02_62V2				:sValveVisu; 			(* ISK Vereinzeler ein-/ausfahren*)
	ST02_62_Y4   			:sValveVisu; 			(*ST02_62_Y4 Kamera Ausschleusen Bandstrecke (Valve) *)

	ST02_35Y01 			:sValveVisu; 			(*1: Einschaltventil Hauptluft Tampondruckanlage*)

	ST02_FDB_54_B41		:sDigInVisu; (* Kamera ISK anwesend an Prüfposition *)

	ST02_DT_65B11  		:sDigInVisu; (* Tampondrucker Nest 1 leer *)
	ST02_DT_65B21  		:sDigInVisu; (* Tampondrucker Nest 2 leer *)

	ST03_51_M1 			: sDigInVisu; (* Bandmotor *)
	ST03_60_M1 			: sDigInVisu; (* Bandmotor Prüfteile *)


(*---------------------------------------------------------------------------
  Station03
  ---------------------------------------------------------------------------*)
	ST03_125_F1 		: sDigInVisu; (* Absicherung Roboter iO *)
	Robot01					:	sEpsonRobotVisu;

	St03_120_A1_A14: sDigInVisu;(*Roboter opt.- Tool 2 ist ein*)
	ST03_400_B12_6 : sDigInVisu; (* Schwenkmodul AST (Roboterkopf) *)
	ST03_400_B12_7 : sDigInVisu; (* Schwenkmodul GST (Roboterkopf) *)
	ST03_400_B54_7: sDigInVisu; (* Tray Testteile in Position *)
	ST03_8_75_B13_5: sDigInVisu; (*voll/belegt keine Prüfmittel mehr*)
	ST03_8_75_B13_6: sDigInVisu; (*belegt mit 6 Prüfmittel*)
	ST03_BG3_X53_0:	sDigOutInVisu; (*Taster Start Band Dummyprüfung*)
	ST03_A5 : sDigOutInVisu; (* Förderbandmotor Oriental *)
	ST03_601V1_A1 : sDigOutInVisu; (* FörderbandPrüfteile *)
	ST03_V2	: sDigInVisu; (* Störung Motor Förderband Oriental *)

